ABB RAPID module: 000F2625

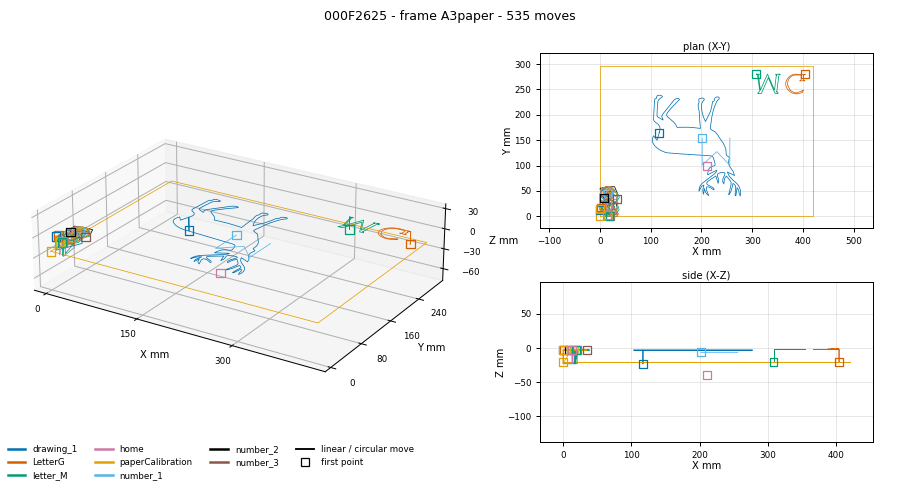
[picture p0: tool path of 000F2625 in frame A3paper, 535 of 535 moves have a stored position in this frame; points joined in program order, loops and branches not executed]
MODULE Module1
	CONST robtarget Target_960:=[[114.097930092,195.477622506,-57.989262096],[0.296983382,-0.000000027,0.000000028,0.954882648],[-1,-1,2,0],[9E+09,9E+09,9E+09,9E+09,9E+09,9E+09]];
	CONST robtarget Target_970:=[[308,280,-20],[1,0,0,0],[0,0,0,0],[9E+09,9E+09,9E+09,9E+09,9E+09,9E+09]];
	CONST robtarget Target_980:=[[308,280,-1],[1,0,0,0],[0,0,0,0],[9E+09,9E+09,9E+09,9E+09,9E+09,9E+09]];
	CONST robtarget Target_990:=[[308,279.6,-1],[1,0,0,0],[0,0,0,0],[9E+09,9E+09,9E+09,9E+09,9E+09,9E+09]];
	CONST robtarget Target_1000:=[[309.6,279.3,-1],[1,0,0,0],[0,0,0,0],[9E+09,9E+09,9E+09,9E+09,9E+09,9E+09]];
	CONST robtarget Target_1010:=[[310.2,278.4,-1],[1,0,0,0],[0,0,0,0],[9E+09,9E+09,9E+09,9E+09,9E+09,9E+09]];
	CONST robtarget Target_1020:=[[314.9,246.9,-1],[1,0,0,0],[0,0,2,0],[9E+09,9E+09,9E+09,9E+09,9E+09,9E+09]];
	CONST robtarget Target_1040:=[[310.75,242.39,-1],[1,0,0,0],[0,0,2,0],[9E+09,9E+09,9E+09,9E+09,9E+09,9E+09]];
	CONST robtarget Target_1050:=[[310.75,241.99,-1],[1,0,0,0],[0,0,0,0],[9E+09,9E+09,9E+09,9E+09,9E+09,9E+09]];
	CONST robtarget Target_1060:=[[317.99,241.99,-1],[1,0,0,0],[0,0,0,0],[9E+09,9E+09,9E+09,9E+09,9E+09,9E+09]];
	CONST robtarget Target_1070:=[[331.45,273.1,-1],[1,0,0,0],[0,0,0,0],[9E+09,9E+09,9E+09,9E+09,9E+09,9E+09]];
	CONST robtarget Target_1080:=[[344.92,241.99,-1],[1,0,0,0],[0,0,0,0],[9E+09,9E+09,9E+09,9E+09,9E+09,9E+09]];
	CONST robtarget Target_1090:=[[351,241.99,-1],[1,0,0,0],[0,0,0,0],[9E+09,9E+09,9E+09,9E+09,9E+09,9E+09]];
	CONST robtarget Target_1100:=[[351,242.39,-1],[1,0,0,0],[0,0,0,0],[9E+09,9E+09,9E+09,9E+09,9E+09,9E+09]];
	CONST robtarget Target_1110:=[[348.2,244.8,-1],[1,0,0,0],[0,0,0,0],[9E+09,9E+09,9E+09,9E+09,9E+09,9E+09]];
	CONST robtarget Target_1120:=[[347.98,246,-1],[1,0,0,0],[0,0,0,0],[9E+09,9E+09,9E+09,9E+09,9E+09,9E+09]];
	CONST robtarget Target_1130:=[[352.51,278,-1],[1,0,0,0],[0,0,0,0],[9E+09,9E+09,9E+09,9E+09,9E+09,9E+09]];
	CONST robtarget Target_1140:=[[353,279,-1],[1,0,0,0],[0,0,0,0],[9E+09,9E+09,9E+09,9E+09,9E+09,9E+09]];
	CONST robtarget Target_1150:=[[354.8,279.7,-1],[1,0,0,0],[0,0,0,0],[9E+09,9E+09,9E+09,9E+09,9E+09,9E+09]];
	CONST robtarget Target_1160:=[[354.8,280,-1],[1,0,0,0],[0,0,0,0],[9E+09,9E+09,9E+09,9E+09,9E+09,9E+09]];
	CONST robtarget Target_1170:=[[346.2,280,-1],[1,0,0,0],[0,0,0,0],[9E+09,9E+09,9E+09,9E+09,9E+09,9E+09]];
	CONST robtarget Target_1180:=[[346.2,279.7,-1],[1,0,0,0],[0,0,0,0],[9E+09,9E+09,9E+09,9E+09,9E+09,9E+09]];
	CONST robtarget Target_1190:=[[347.51,279.3,-1],[1,0,0,0],[0,0,0,0],[9E+09,9E+09,9E+09,9E+09,9E+09,9E+09]];
	CONST robtarget Target_1200:=[[347.96,278,-1],[1,0,0,0],[0,0,0,0],[9E+09,9E+09,9E+09,9E+09,9E+09,9E+09]];
	CONST robtarget Target_1210:=[[343.88,248.52,-1],[1,0,0,0],[0,0,0,0],[9E+09,9E+09,9E+09,9E+09,9E+09,9E+09]];
	CONST robtarget Target_1220:=[[330.1,280,-1],[1,0,0,0],[0,0,0,0],[9E+09,9E+09,9E+09,9E+09,9E+09,9E+09]];
	CONST robtarget Target_1230:=[[329.81,280,-1],[1,0,0,0],[0,0,0,0],[9E+09,9E+09,9E+09,9E+09,9E+09,9E+09]];
	CONST robtarget Target_1240:=[[316.05,248.51,-1],[1,0,0,0],[0,0,0,0],[9E+09,9E+09,9E+09,9E+09,9E+09,9E+09]];
	CONST robtarget Target_1250:=[[312.1,278,-1],[1,0,0,0],[0,0,0,0],[9E+09,9E+09,9E+09,9E+09,9E+09,9E+09]];
	CONST robtarget Target_1260:=[[312.3,279,-1],[1,0,0,0],[0,0,0,0],[9E+09,9E+09,9E+09,9E+09,9E+09,9E+09]];
	CONST robtarget Target_1270:=[[313.8,279.7,-1],[1,0,0,0],[0,0,0,0],[9E+09,9E+09,9E+09,9E+09,9E+09,9E+09]];
	CONST robtarget Target_1280:=[[313.8,280,-1],[1,0,0,0],[0,0,0,0],[9E+09,9E+09,9E+09,9E+09,9E+09,9E+09]];
	CONST robtarget Target_1290:=[[308,280,-1],[1,0,0,0],[0,0,0,0],[9E+09,9E+09,9E+09,9E+09,9E+09,9E+09]];
	CONST robtarget Target_1300:=[[308,280,-20],[1,0,0,0],[0,0,0,0],[9E+09,9E+09,9E+09,9E+09,9E+09,9E+09]];
	CONST robtarget Target_1310:=[[403.47,280,-20],[1,0,0,0],[0,0,0,0],[9E+09,9E+09,9E+09,9E+09,9E+09,9E+09]];
	CONST robtarget Target_1320:=[[403.47,280,-1],[1,0,0,0],[0,0,1,0],[9E+09,9E+09,9E+09,9E+09,9E+09,9E+09]];
	CONST robtarget Target_1330:=[[387,280,-1],[1,0,0,0],[0,0,1,0],[9E+09,9E+09,9E+09,9E+09,9E+09,9E+09]];
	CONST robtarget Target_1340:=[[365.71,260,-1],[1,0,0,0],[0,0,1,0],[9E+09,9E+09,9E+09,9E+09,9E+09,9E+09]];
	CONST robtarget Target_1350:=[[382,241.9,-1],[1,0,0,0],[0,0,1,0],[9E+09,9E+09,9E+09,9E+09,9E+09,9E+09]];
	CONST robtarget Target_1360:=[[387,241.3,-1],[1,0,0,0],[0,0,1,0],[9E+09,9E+09,9E+09,9E+09,9E+09,9E+09]];
	CONST robtarget Target_1370:=[[398.5,244.5,-1],[1,0,0,0],[0,0,1,0],[9E+09,9E+09,9E+09,9E+09,9E+09,9E+09]];
	CONST robtarget Target_1380:=[[400.8,248.26,-1],[1,0,0,0],[0,0,1,0],[9E+09,9E+09,9E+09,9E+09,9E+09,9E+09]];
	CONST robtarget Target_1390:=[[400.4,248.26,-1],[1,0,0,0],[0,0,1,0],[9E+09,9E+09,9E+09,9E+09,9E+09,9E+09]];
	CONST robtarget Target_1400:=[[387,242.79,-1],[1,0,0,0],[0,0,1,0],[9E+09,9E+09,9E+09,9E+09,9E+09,9E+09]];
	CONST robtarget Target_1410:=[[382,244.2,-1],[1,0,0,0],[0,0,1,0],[9E+09,9E+09,9E+09,9E+09,9E+09,9E+09]];
	CONST robtarget Target_1420:=[[370,258,-1],[1,0,0,0],[0,0,1,0],[9E+09,9E+09,9E+09,9E+09,9E+09,9E+09]];
	CONST robtarget Target_1420A:=[[380,272,-1],[1,0,0,0],[0,0,1,0],[9E+09,9E+09,9E+09,9E+09,9E+09,9E+09]];
	CONST robtarget Target_1430:=[[388,278.4,-1],[1,0,0,0],[0,0,1,0],[9E+09,9E+09,9E+09,9E+09,9E+09,9E+09]];
	CONST robtarget Target_1440:=[[392,278.99,-1],[1,0,0,0],[0,0,1,0],[9E+09,9E+09,9E+09,9E+09,9E+09,9E+09]];
	CONST robtarget Target_1450:=[[393,278.75,-1],[1,0,0,0],[0,0,1,0],[9E+09,9E+09,9E+09,9E+09,9E+09,9E+09]];
	CONST robtarget Target_1460:=[[395.8,278,-1],[1,0,0,0],[0,0,1,0],[9E+09,9E+09,9E+09,9E+09,9E+09,9E+09]];
	CONST robtarget Target_1470:=[[396.3,276,-1],[1,0,0,0],[0,0,1,0],[9E+09,9E+09,9E+09,9E+09,9E+09,9E+09]];
	CONST robtarget Target_1480:=[[392.7,278.3,-1],[1,0,0,0],[0,0,1,0],[9E+09,9E+09,9E+09,9E+09,9E+09,9E+09]];
	CONST robtarget Target_1490:=[[395.7,278.2,-1],[1,0,0,0],[0,0,1,0],[9E+09,9E+09,9E+09,9E+09,9E+09,9E+09]];
	CONST robtarget Target_1500:=[[396.3,276,-1],[1,0,0,0],[0,0,1,0],[9E+09,9E+09,9E+09,9E+09,9E+09,9E+09]];
	CONST robtarget Target_1510:=[[396.3,269.1,-1],[1,0,0,0],[0,0,1,0],[9E+09,9E+09,9E+09,9E+09,9E+09,9E+09]];
	CONST robtarget Target_1520:=[[394.9,267.9,-1],[1,0,0,0],[0,0,1,0],[9E+09,9E+09,9E+09,9E+09,9E+09,9E+09]];
	CONST robtarget Target_1530:=[[393.51,267.1,-1],[1,0,0,0],[0,0,1,0],[9E+09,9E+09,9E+09,9E+09,9E+09,9E+09]];
	CONST robtarget Target_1540:=[[393.5,266.8,-1],[1,0,0,0],[0,0,1,0],[9E+09,9E+09,9E+09,9E+09,9E+09,9E+09]];
	CONST robtarget Target_1550:=[[403.5,266.8,-1],[1,0,0,0],[0,0,1,0],[9E+09,9E+09,9E+09,9E+09,9E+09,9E+09]];
	CONST robtarget Target_1560:=[[403.5,267.1,-1],[1,0,0,0],[0,0,1,0],[9E+09,9E+09,9E+09,9E+09,9E+09,9E+09]];
	CONST robtarget Target_1570:=[[401.2,267.9,-1],[1,0,0,0],[0,0,1,0],[9E+09,9E+09,9E+09,9E+09,9E+09,9E+09]];
	CONST robtarget Target_1580:=[[400.8,269.1,-1],[1,0,0,0],[0,0,1,0],[9E+09,9E+09,9E+09,9E+09,9E+09,9E+09]];
	CONST robtarget Target_1590:=[[400.8,276,-1],[1,0,0,0],[0,0,1,0],[9E+09,9E+09,9E+09,9E+09,9E+09,9E+09]];
	CONST robtarget Target_1600:=[[401.2,279,-1],[1,0,0,0],[0,0,1,0],[9E+09,9E+09,9E+09,9E+09,9E+09,9E+09]];
	CONST robtarget Target_1610:=[[403.5,279.7,-1],[1,0,0,0],[0,0,1,0],[9E+09,9E+09,9E+09,9E+09,9E+09,9E+09]];
	CONST robtarget Target_1630:=[[210,100,-40],[1,0,0,0],[0,0,0,0],[9E+09,9E+09,9E+09,9E+09,9E+09,9E+09]];
	CONST robtarget image_startTarget:=[[114.097941212,195.477543406,-3],[0.296983386,0,0,0.954882646],[-1,0,2,0],[9E+09,9E+09,9E+09,9E+09,9E+09,9E+09]];
	CONST robtarget Target_1421:=[[374.2,273.2,-1],[1,0,0,0],[0,0,1,0],[9E+09,9E+09,9E+09,9E+09,9E+09,9E+09]];
	CONST robtarget Target_1411:=[[374.3,249.1,-1],[1,0,0,0],[0,0,1,0],[9E+09,9E+09,9E+09,9E+09,9E+09,9E+09]];
	CONST robtarget Target_1331:=[[370.8,273,-1],[1,0,0,0],[0,0,1,0],[9E+09,9E+09,9E+09,9E+09,9E+09,9E+09]];
	CONST robtarget Target_1341:=[[372.4,247,-1],[1,0,0,0],[0,0,1,0],[9E+09,9E+09,9E+09,9E+09,9E+09,9E+09]];
	CONST robtarget Target_1620:=[[403.5,280,-1],[1,0,0,0],[0,0,1,0],[9E+09,9E+09,9E+09,9E+09,9E+09,9E+09]];
    CONST robtarget Target_2160:=[[193.370337383,219.913130465,-3],[1,0,0,0],[0,0,0,0],[9E+09,9E+09,9E+09,9E+09,9E+09,9E+09]];
    CONST robtarget Target_2190:=[[195.261015335,231.205877786,-3],[1,0,0,0],[0,0,0,0],[9E+09,9E+09,9E+09,9E+09,9E+09,9E+09]];
    CONST robtarget Target_2240:=[[202.476909017,225.935782034,-3],[1,0,0,0],[0,0,0,0],[9E+09,9E+09,9E+09,9E+09,9E+09,9E+09]];
    CONST robtarget Target_2250:=[[200.458270111,222.059210742,-3],[1,0,0,0],[0,0,0,0],[9E+09,9E+09,9E+09,9E+09,9E+09,9E+09]];
    CONST robtarget Target_2260:=[[200.131870923,213.002260799,-3],[1,0,0,0],[0,0,0,0],[9E+09,9E+09,9E+09,9E+09,9E+09,9E+09]];
    CONST robtarget Target_2270:=[[201.352548333,204.144326867,-3],[1,0,0,0],[0,0,0,0],[9E+09,9E+09,9E+09,9E+09,9E+09,9E+09]];
    CONST robtarget Target_2280:=[[203.989899977,195.415486359,-3],[1,0,0,0],[0,0,0,0],[9E+09,9E+09,9E+09,9E+09,9E+09,9E+09]];
    CONST robtarget Target_2310:=[[219.57359463,213.353914551,-3],[1,0,0,0],[0,0,0,0],[9E+09,9E+09,9E+09,9E+09,9E+09,9E+09]];
    CONST robtarget Target_2320:=[[221.72168992,225.083729881,-3],[1,0,0,0],[0,0,0,0],[9E+09,9E+09,9E+09,9E+09,9E+09,9E+09]];
    CONST robtarget Target_2370:=[[226.65209234,233.190693627,-3],[1,0,0,0],[0,0,0,0],[9E+09,9E+09,9E+09,9E+09,9E+09,9E+09]];
    CONST robtarget Target_2440:=[[229.869479521,225.835975339,-3],[1,0,0,0],[0,0,0,0],[9E+09,9E+09,9E+09,9E+09,9E+09,9E+09]];
    CONST robtarget Target_2450:=[[227.167304938,219.606802526,-3],[1,0,0,0],[0,0,0,0],[9E+09,9E+09,9E+09,9E+09,9E+09,9E+09]];
    CONST robtarget Target_2470:=[[220.688053949,197.559828522,-3],[1,0,0,0],[0,0,0,0],[9E+09,9E+09,9E+09,9E+09,9E+09,9E+09]];
    CONST robtarget Target_2490:=[[217.906200407,171.90434605,-3],[1,0,0,0],[0,0,0,0],[9E+09,9E+09,9E+09,9E+09,9E+09,9E+09]];
    CONST robtarget Target_2510:=[[227.578391856,165.853990796,-3],[1,0,0,0],[0,0,0,0],[9E+09,9E+09,9E+09,9E+09,9E+09,9E+09]];
    CONST robtarget Target_2520:=[[232.79626775,159.200927161,-3],[1,0,0,0],[0,0,0,0],[9E+09,9E+09,9E+09,9E+09,9E+09,9E+09]];
    CONST robtarget Target_2530:=[[235.197557217,154.8951234,-3],[1,0,0,0],[0,0,0,0],[9E+09,9E+09,9E+09,9E+09,9E+09,9E+09]];
    CONST robtarget Target_2560:=[[248.128216692,130.946667408,-3],[1,0,0,0],[0,0,0,0],[9E+09,9E+09,9E+09,9E+09,9E+09,9E+09]];
    CONST robtarget Target_2580:=[[249.072498858,120.410096923,-3],[1,0,0,0],[0,0,0,0],[9E+09,9E+09,9E+09,9E+09,9E+09,9E+09]];
    CONST robtarget Target_2590:=[[251.497695182,118.536506038,-3],[1,0,0,0],[0,0,0,0],[9E+09,9E+09,9E+09,9E+09,9E+09,9E+09]];
    CONST robtarget Target_2610:=[[254.693387483,115.452076001,-3],[1,0,0,0],[0,0,0,0],[9E+09,9E+09,9E+09,9E+09,9E+09,9E+09]];
    CONST robtarget Target_2660:=[[265.141029781,80.351141961,-3],[1,0,0,0],[0,0,0,0],[9E+09,9E+09,9E+09,9E+09,9E+09,9E+09]];
    CONST robtarget Target_2680:=[[253.43619882,81.678122788,-3],[1,0,0,0],[0,0,0,0],[9E+09,9E+09,9E+09,9E+09,9E+09,9E+09]];
    CONST robtarget Target_2690:=[[256.347942609,77.175605659,-3],[1,0,0,0],[0,0,0,0],[9E+09,9E+09,9E+09,9E+09,9E+09,9E+09]];
    CONST robtarget Target_2710:=[[267.614835775,66.494604603,-3],[1,0,0,0],[0,0,0,0],[9E+09,9E+09,9E+09,9E+09,9E+09,9E+09]];
    CONST robtarget Target_2720:=[[271.684226977,62.292746796,-3],[1,0,0,0],[0,0,0,0],[9E+09,9E+09,9E+09,9E+09,9E+09,9E+09]];
    CONST robtarget Target_2730:=[[274.598698271,57.568830631,-3],[1,0,0,0],[0,0,0,0],[9E+09,9E+09,9E+09,9E+09,9E+09,9E+09]];
    CONST robtarget Target_2740:=[[276.417527718,52.342499268,-3],[1,0,0,0],[0,0,0,0],[9E+09,9E+09,9E+09,9E+09,9E+09,9E+09]];
    CONST robtarget Target_2750:=[[277.199993374,46.633395866,-3],[1,0,0,0],[0,0,0,0],[9E+09,9E+09,9E+09,9E+09,9E+09,9E+09]];
    CONST robtarget Target_2760:=[[276.903780142,43.337729466,-3],[1,0,0,0],[0,0,0,0],[9E+09,9E+09,9E+09,9E+09,9E+09,9E+09]];
    CONST robtarget Target_2770:=[[276.283936631,40.026597635,-3],[1,0,0,0],[0,0,0,0],[9E+09,9E+09,9E+09,9E+09,9E+09,9E+09]];
    CONST robtarget Target_2780:=[[274.453452076,43.865061405,-3],[1,0,0,0],[0,0,0,0],[9E+09,9E+09,9E+09,9E+09,9E+09,9E+09]];
    CONST robtarget Target_2790:=[[273.824145046,48.089825742,-3],[1,0,0,0],[0,0,0,0],[9E+09,9E+09,9E+09,9E+09,9E+09,9E+09]];
    CONST robtarget Target_2810:=[[270.016935967,56.440062852,-3],[1,0,0,0],[0,0,0,0],[9E+09,9E+09,9E+09,9E+09,9E+09,9E+09]];
    CONST robtarget Target_2820:=[[267.749530853,40.667201266,-3],[1,0,0,0],[0,0,0,0],[9E+09,9E+09,9E+09,9E+09,9E+09,9E+09]];
    CONST robtarget Target_2830:=[[266.302922269,40.756977809,-3],[1,0,0,0],[0,0,0,0],[9E+09,9E+09,9E+09,9E+09,9E+09,9E+09]];
    CONST robtarget Target_2840:=[[266.441249646,47.650430951,-3],[1,0,0,0],[0,0,0,0],[9E+09,9E+09,9E+09,9E+09,9E+09,9E+09]];
    CONST robtarget Target_2850:=[[267.430396017,57.809270006,-3],[1,0,0,0],[0,0,0,0],[9E+09,9E+09,9E+09,9E+09,9E+09,9E+09]];
    CONST robtarget Target_2860:=[[266.669716785,60.560651269,-3],[1,0,0,0],[0,0,0,0],[9E+09,9E+09,9E+09,9E+09,9E+09,9E+09]];
    CONST robtarget Target_2870:=[[264.903208645,62.848641641,-3],[1,0,0,0],[0,0,0,0],[9E+09,9E+09,9E+09,9E+09,9E+09,9E+09]];
    CONST robtarget Target_2880:=[[262.176964385,64.847561878,-3],[1,0,0,0],[0,0,0,0],[9E+09,9E+09,9E+09,9E+09,9E+09,9E+09]];
    CONST robtarget Target_2890:=[[259.299549793,53.075582965,-3],[1,0,0,0],[0,0,0,0],[9E+09,9E+09,9E+09,9E+09,9E+09,9E+09]];
    CONST robtarget Target_2910:=[[253.896826863,42.44360071,-3],[1,0,0,0],[0,0,0,0],[9E+09,9E+09,9E+09,9E+09,9E+09,9E+09]];
    CONST robtarget Target_2920:=[[253.921604349,44.335351342,-3],[1,0,0,0],[0,0,0,0],[9E+09,9E+09,9E+09,9E+09,9E+09,9E+09]];
    CONST robtarget Target_2930:=[[258.274708163,62.583521728,-3],[1,0,0,0],[0,0,0,0],[9E+09,9E+09,9E+09,9E+09,9E+09,9E+09]];
    CONST robtarget Target_2940:=[[258.451861421,65.72308068,-3],[1,0,0,0],[0,0,0,0],[9E+09,9E+09,9E+09,9E+09,9E+09,9E+09]];
    CONST robtarget Target_2950:=[[257.604969868,68.580619068,-3],[1,0,0,0],[0,0,0,0],[9E+09,9E+09,9E+09,9E+09,9E+09,9E+09]];
    CONST robtarget Target_2960:=[[253.567432927,74.071600383,-3],[1,0,0,0],[0,0,0,0],[9E+09,9E+09,9E+09,9E+09,9E+09,9E+09]];
    CONST robtarget Target_2970:=[[249.243881242,79.371580046,-3],[1,0,0,0],[0,0,0,0],[9E+09,9E+09,9E+09,9E+09,9E+09,9E+09]];
    CONST robtarget Target_2980:=[[246.352038922,75.978183413,-3],[1,0,0,0],[0,0,0,0],[9E+09,9E+09,9E+09,9E+09,9E+09,9E+09]];
    CONST robtarget Target_2990:=[[244.977183436,72.142467996,-3],[1,0,0,0],[0,0,0,0],[9E+09,9E+09,9E+09,9E+09,9E+09,9E+09]];
    CONST robtarget Target_3010:=[[242.513799023,66.424388789,-3],[1,0,0,0],[0,0,0,0],[9E+09,9E+09,9E+09,9E+09,9E+09,9E+09]];
    CONST robtarget Target_3030:=[[242.453890553,75.021110222,-3],[1,0,0,0],[0,0,0,0],[9E+09,9E+09,9E+09,9E+09,9E+09,9E+09]];
    CONST robtarget Target_3040:=[[245.184309174,80.346921596,-3],[1,0,0,0],[0,0,0,0],[9E+09,9E+09,9E+09,9E+09,9E+09,9E+09]];
    CONST robtarget Target_3050:=[[246.355111707,84.063986783,-3],[1,0,0,0],[0,0,0,0],[9E+09,9E+09,9E+09,9E+09,9E+09,9E+09]];
    CONST robtarget Target_3060:=[[245.799291444,85.605935054,-3],[1,0,0,0],[0,0,0,0],[9E+09,9E+09,9E+09,9E+09,9E+09,9E+09]];
    CONST robtarget Target_3070:=[[243.989820642,86.456427668,-3],[1,0,0,0],[0,0,0,0],[9E+09,9E+09,9E+09,9E+09,9E+09,9E+09]];
    CONST robtarget Target_3080:=[[238.686656522,86.356933008,-3],[1,0,0,0],[0,0,0,0],[9E+09,9E+09,9E+09,9E+09,9E+09,9E+09]];
    CONST robtarget Target_3090:=[[233.626373536,84.723508323,-3],[1,0,0,0],[0,0,0,0],[9E+09,9E+09,9E+09,9E+09,9E+09,9E+09]];
    CONST robtarget Target_3110:=[[231.229705834,80.92138457,-3],[1,0,0,0],[0,0,0,0],[9E+09,9E+09,9E+09,9E+09,9E+09,9E+09]];
    CONST robtarget Target_3120:=[[232.687410286,76.08625905,-3],[1,0,0,0],[0,0,0,0],[9E+09,9E+09,9E+09,9E+09,9E+09,9E+09]];
    CONST robtarget Target_3130:=[[233.844814545,70.463867465,-3],[1,0,0,0],[0,0,0,0],[9E+09,9E+09,9E+09,9E+09,9E+09,9E+09]];
    CONST robtarget Target_3140:=[[232.683868526,64.986793847,-3],[1,0,0,0],[0,0,0,0],[9E+09,9E+09,9E+09,9E+09,9E+09,9E+09]];
    CONST robtarget Target_3150:=[[228.374978172,79.484110725,-3],[1,0,0,0],[0,0,0,0],[9E+09,9E+09,9E+09,9E+09,9E+09,9E+09]];
    CONST robtarget Target_3160:=[[219.965736687,74.015207284,-3],[1,0,0,0],[0,0,0,0],[9E+09,9E+09,9E+09,9E+09,9E+09,9E+09]];
    CONST robtarget Target_3170:=[[212.554359432,68.787624505,-3],[1,0,0,0],[0,0,0,0],[9E+09,9E+09,9E+09,9E+09,9E+09,9E+09]];
    CONST robtarget Target_3180:=[[210.677030599,66.626673914,-3],[1,0,0,0],[0,0,0,0],[9E+09,9E+09,9E+09,9E+09,9E+09,9E+09]];
    CONST robtarget Target_3190:=[[210.38708356,64.517394422,-3],[1,0,0,0],[0,0,0,0],[9E+09,9E+09,9E+09,9E+09,9E+09,9E+09]];
    CONST robtarget Target_3210:=[[214.11130813,61.047061647,-3],[1,0,0,0],[0,0,0,0],[9E+09,9E+09,9E+09,9E+09,9E+09,9E+09]];
    CONST robtarget Target_3220:=[[222.416533213,56.844968834,-3],[1,0,0,0],[0,0,0,0],[9E+09,9E+09,9E+09,9E+09,9E+09,9E+09]];
    CONST robtarget Target_3230:=[[223.832262364,55.151481233,-3],[1,0,0,0],[0,0,0,0],[9E+09,9E+09,9E+09,9E+09,9E+09,9E+09]];
    CONST robtarget Target_3240:=[[224.991497966,53.059964778,-3],[1,0,0,0],[0,0,0,0],[9E+09,9E+09,9E+09,9E+09,9E+09,9E+09]];
    CONST robtarget Target_3260:=[[217.660699108,56.478310873,-3],[1,0,0,0],[0,0,0,0],[9E+09,9E+09,9E+09,9E+09,9E+09,9E+09]];
    CONST robtarget Target_3270:=[[214.198336017,57.976316513,-3],[1,0,0,0],[0,0,0,0],[9E+09,9E+09,9E+09,9E+09,9E+09,9E+09]];
    CONST robtarget Target_3280:=[[210.117558581,57.951519862,-3],[1,0,0,0],[0,0,0,0],[9E+09,9E+09,9E+09,9E+09,9E+09,9E+09]];
    CONST robtarget Target_3290:=[[209.641800543,53.313049599,-3],[1,0,0,0],[0,0,0,0],[9E+09,9E+09,9E+09,9E+09,9E+09,9E+09]];
    CONST robtarget Target_3310:=[[214.391838304,40.955022791,-3],[1,0,0,0],[0,0,0,0],[9E+09,9E+09,9E+09,9E+09,9E+09,9E+09]];
    CONST robtarget Target_3320:=[[210.799968866,43.482482486,-3],[1,0,0,0],[0,0,0,0],[9E+09,9E+09,9E+09,9E+09,9E+09,9E+09]];
    CONST robtarget Target_3330:=[[208.378326367,46.710824702,-3],[1,0,0,0],[0,0,0,0],[9E+09,9E+09,9E+09,9E+09,9E+09,9E+09]];
    CONST robtarget Target_3340:=[[205.519567882,54.640553293,-3],[1,0,0,0],[0,0,0,0],[9E+09,9E+09,9E+09,9E+09,9E+09,9E+09]];
    CONST robtarget Target_3350:=[[204.274957824,43.449915608,-3],[1,0,0,0],[0,0,0,0],[9E+09,9E+09,9E+09,9E+09,9E+09,9E+09]];
    CONST robtarget Target_3360:=[[202.779864784,47.961332689,-3],[1,0,0,0],[0,0,0,0],[9E+09,9E+09,9E+09,9E+09,9E+09,9E+09]];
    CONST robtarget Target_3370:=[[202.686470534,52.473353811,-3],[1,0,0,0],[0,0,0,0],[9E+09,9E+09,9E+09,9E+09,9E+09,9E+09]];
    CONST robtarget Target_3380:=[[204.779738543,61.691960466,-3],[1,0,0,0],[0,0,0,0],[9E+09,9E+09,9E+09,9E+09,9E+09,9E+09]];
    CONST robtarget Target_3390:=[[200.828885863,59.46054831,-3],[1,0,0,0],[0,0,0,0],[9E+09,9E+09,9E+09,9E+09,9E+09,9E+09]];
    CONST robtarget Target_3410:=[[195.145559108,49.337942562,-3],[1,0,0,0],[0,0,0,0],[9E+09,9E+09,9E+09,9E+09,9E+09,9E+09]];
    CONST robtarget Target_3420:=[[195.353663461,54.280625926,-3],[1,0,0,0],[0,0,0,0],[9E+09,9E+09,9E+09,9E+09,9E+09,9E+09]];
    CONST robtarget Target_3430:=[[196.676958422,58.695618887,-3],[1,0,0,0],[0,0,0,0],[9E+09,9E+09,9E+09,9E+09,9E+09,9E+09]];
    CONST robtarget Target_3440:=[[199.103095305,62.59104984,-3],[1,0,0,0],[0,0,0,0],[9E+09,9E+09,9E+09,9E+09,9E+09,9E+09]];
    CONST robtarget Target_3450:=[[202.619725421,65.975047185,-3],[1,0,0,0],[0,0,0,0],[9E+09,9E+09,9E+09,9E+09,9E+09,9E+09]];
    CONST robtarget Target_3470:=[[228.146134612,86.522665975,-3],[1,0,0,0],[0,0,0,0],[9E+09,9E+09,9E+09,9E+09,9E+09,9E+09]];
    CONST robtarget Target_3480:=[[230.400867961,89.633137216,-3],[1,0,0,0],[0,0,0,0],[9E+09,9E+09,9E+09,9E+09,9E+09,9E+09]];
    CONST robtarget Target_3490:=[[229.502924222,90.649093077,-3],[1,0,0,0],[0,0,0,0],[9E+09,9E+09,9E+09,9E+09,9E+09,9E+09]];
    CONST robtarget Target_3510:=[[213.02947803,88.518895223,-3],[1,0,0,0],[0,0,0,0],[9E+09,9E+09,9E+09,9E+09,9E+09,9E+09]];
    CONST robtarget Target_3520:=[[214.278806706,92.822596592,-3],[1,0,0,0],[0,0,0,0],[9E+09,9E+09,9E+09,9E+09,9E+09,9E+09]];
    CONST robtarget Target_3530:=[[216.417539352,95.955068284,-3],[1,0,0,0],[0,0,0,0],[9E+09,9E+09,9E+09,9E+09,9E+09,9E+09]];
    CONST robtarget Target_3540:=[[219.585437503,98.050973568,-3],[1,0,0,0],[0,0,0,0],[9E+09,9E+09,9E+09,9E+09,9E+09,9E+09]];
    CONST robtarget Target_3550:=[[223.922262697,99.244975714,-3],[1,0,0,0],[0,0,0,0],[9E+09,9E+09,9E+09,9E+09,9E+09,9E+09]];
    CONST robtarget Target_3560:=[[226.759287881,100.694337329,-3],[1,0,0,0],[0,0,0,0],[9E+09,9E+09,9E+09,9E+09,9E+09,9E+09]];
    CONST robtarget Target_3570:=[[226.681756776,103.944262165,-3],[1,0,0,0],[0,0,0,0],[9E+09,9E+09,9E+09,9E+09,9E+09,9E+09]];
    CONST robtarget Target_3580:=[[224.505103701,112.138872075,-3],[1,0,0,0],[0,0,0,0],[9E+09,9E+09,9E+09,9E+09,9E+09,9E+09]];
    CONST robtarget Target_3590:=[[223.414408001,115.469817817,-3],[1,0,0,0],[0,0,0,0],[9E+09,9E+09,9E+09,9E+09,9E+09,9E+09]];
    CONST robtarget Target_3610:=[[219.460026303,118.825512034,-3],[1,0,0,0],[0,0,0,0],[9E+09,9E+09,9E+09,9E+09,9E+09,9E+09]];
    CONST robtarget Target_3620:=[[215.936165455,119.356824487,-3],[1,0,0,0],[0,0,0,0],[9E+09,9E+09,9E+09,9E+09,9E+09,9E+09]];
    CONST robtarget Target_3630:=[[155.66830507,123.260946897,-3],[1,0,0,0],[0,0,0,0],[9E+09,9E+09,9E+09,9E+09,9E+09,9E+09]];
    CONST robtarget Target_3640:=[[133.585682803,125.008606143,-3],[1,0,0,0],[0,0,0,0],[9E+09,9E+09,9E+09,9E+09,9E+09,9E+09]];
    CONST robtarget Target_3650:=[[128.099986881,126.297578543,-3],[1,0,0,0],[0,0,0,0],[9E+09,9E+09,9E+09,9E+09,9E+09,9E+09]];
    CONST robtarget Target_3660:=[[122.770725675,128.44117716,-3],[1,0,0,0],[0,0,0,0],[9E+09,9E+09,9E+09,9E+09,9E+09,9E+09]];
    CONST robtarget Target_3670:=[[118.375825136,130.605132148,-3],[1,0,0,0],[0,0,0,0],[9E+09,9E+09,9E+09,9E+09,9E+09,9E+09]];
    CONST robtarget Target_3680:=[[114.276287738,133.278163879,-3],[1,0,0,0],[0,0,0,0],[9E+09,9E+09,9E+09,9E+09,9E+09,9E+09]];
    CONST robtarget Target_3690:=[[108.31401898,138.447566871,-3],[1,0,0,0],[0,0,0,0],[9E+09,9E+09,9E+09,9E+09,9E+09,9E+09]];
    CONST robtarget Target_3710:=[[103.212048819,150.747792156,-3],[1,0,0,0],[0,0,0,0],[9E+09,9E+09,9E+09,9E+09,9E+09,9E+09]];
    CONST robtarget Target_3720:=[[103.919723158,154.520288699,-3],[1,0,0,0],[0,0,0,0],[9E+09,9E+09,9E+09,9E+09,9E+09,9E+09]];
    CONST robtarget Target_3730:=[[105.613280939,158.670782312,-3],[1,0,0,0],[0,0,0,0],[9E+09,9E+09,9E+09,9E+09,9E+09,9E+09]];
    CONST robtarget Target_3740:=[[112.529465698,149.875319719,-3],[1,0,0,0],[0,0,0,0],[9E+09,9E+09,9E+09,9E+09,9E+09,9E+09]];
    CONST robtarget Target_3750:=[[116.864395565,164.59256718,-3],[1,0,0,0],[0,0,0,0],[9E+09,9E+09,9E+09,9E+09,9E+09,9E+09]];
    CONST robtarget Target_1860:=[[112.780653432,197.331638937,-3],[1,0,0,0],[0,0,0,0],[9E+09,9E+09,9E+09,9E+09,9E+09,9E+09]];
    CONST robtarget Target_2080:=[[152.038829652,175.1593366,-3],[1,0,0,0],[0,0,0,0],[9E+09,9E+09,9E+09,9E+09,9E+09,9E+09]];
    CONST robtarget Target_3020:=[[241.726872614,69.136971847,-3],[1,0,0,0],[0,0,0,0],[9E+09,9E+09,9E+09,9E+09,9E+09,9E+09]];
    CONST robtarget Target_2640:=[[255.55352801,98.15492303,-3],[1,0,0,0],[0,0,0,0],[9E+09,9E+09,9E+09,9E+09,9E+09,9E+09]];
    CONST robtarget Target_2120:=[[197.917101799,173.183120269,-3],[1,0,0,0],[0,0,0,0],[9E+09,9E+09,9E+09,9E+09,9E+09,9E+09]];
    CONST robtarget Target_1850:=[[112.322584565,199.686358994,-3],[1,0,0,0],[0,0,0,0],[9E+09,9E+09,9E+09,9E+09,9E+09,9E+09]];
    CONST robtarget Target_1930:=[[124.987181965,202.815326796,-3],[1,0,0,0],[0,0,0,0],[9E+09,9E+09,9E+09,9E+09,9E+09,9E+09]];
    CONST robtarget Target_1760:=[[113.175108389,237.881718509,-3],[1,0,0,0],[0,0,0,0],[9E+09,9E+09,9E+09,9E+09,9E+09,9E+09]];
    CONST robtarget Target_2570:=[[248.603313012,123.194262198,-3],[1,0,0,0],[0,0,0,0],[9E+09,9E+09,9E+09,9E+09,9E+09,9E+09]];
    CONST robtarget Target_1940:=[[146.479851245,229.690888833,-3],[1,0,0,0],[0,0,0,0],[9E+09,9E+09,9E+09,9E+09,9E+09,9E+09]];
    CONST robtarget Target_1890:=[[124.588660422,189.645922432,-3],[1,0,0,0],[0,0,0,0],[9E+09,9E+09,9E+09,9E+09,9E+09,9E+09]];
    CONST robtarget Target_1990:=[[143.386028726,216.472160161,-3],[1,0,0,0],[0,0,0,0],[9E+09,9E+09,9E+09,9E+09,9E+09,9E+09]];
    CONST robtarget Target_1960:=[[153.996438131,232.359045465,-3],[1,0,0,0],[0,0,0,0],[9E+09,9E+09,9E+09,9E+09,9E+09,9E+09]];
    CONST robtarget Target_1920:=[[122.033123429,198.293656571,-3],[1,0,0,0],[0,0,0,0],[9E+09,9E+09,9E+09,9E+09,9E+09,9E+09]];
    CONST robtarget Target_1970:=[[155.686057122,231.358602968,-3],[1,0,0,0],[0,0,0,0],[9E+09,9E+09,9E+09,9E+09,9E+09,9E+09]];
    CONST robtarget Target_1640:=[[116.864395565,164.59256718,-3],[1,0,0,0],[0,0,0,0],[9E+09,9E+09,9E+09,9E+09,9E+09,9E+09]];
    CONST robtarget Target_1700:=[[105.460399665,190.998170229,-3],[1,0,0,0],[0,0,0,0],[9E+09,9E+09,9E+09,9E+09,9E+09,9E+09]];
    CONST robtarget Target_1800:=[[122.788239246,235.080918952,-3],[1,0,0,0],[0,0,0,0],[9E+09,9E+09,9E+09,9E+09,9E+09,9E+09]];
    CONST robtarget Target_1900:=[[123.322560124,193.264620662,-3],[1,0,0,0],[0,0,0,0],[9E+09,9E+09,9E+09,9E+09,9E+09,9E+09]];
    CONST robtarget Target_2000:=[[138.216503942,210.589237829,-3],[1,0,0,0],[0,0,0,0],[9E+09,9E+09,9E+09,9E+09,9E+09,9E+09]];
    CONST robtarget Target_2100:=[[175.283029198,175.465591704,-3],[1,0,0,0],[0,0,0,0],[9E+09,9E+09,9E+09,9E+09,9E+09,9E+09]];
    CONST robtarget Target_2200:=[[197.204607445,232.112473887,-3],[1,0,0,0],[0,0,0,0],[9E+09,9E+09,9E+09,9E+09,9E+09,9E+09]];
    CONST robtarget Target_2300:=[[216.653373158,204.262410012,-3],[1,0,0,0],[0,0,0,0],[9E+09,9E+09,9E+09,9E+09,9E+09,9E+09]];
    CONST robtarget Target_2400:=[[234.529319608,234.44032996,-3],[1,0,0,0],[0,0,0,0],[9E+09,9E+09,9E+09,9E+09,9E+09,9E+09]];
    CONST robtarget Target_2500:=[[220.374264807,170.158152985,-3],[1,0,0,0],[0,0,0,0],[9E+09,9E+09,9E+09,9E+09,9E+09,9E+09]];
    CONST robtarget Target_2600:=[[253.646962041,117.233560169,-3],[1,0,0,0],[0,0,0,0],[9E+09,9E+09,9E+09,9E+09,9E+09,9E+09]];
    CONST robtarget Target_2700:=[[260.733890497,72.527955155,-3],[1,0,0,0],[0,0,0,0],[9E+09,9E+09,9E+09,9E+09,9E+09,9E+09]];
    CONST robtarget Target_2800:=[[272.857983642,52.38634233,-3],[1,0,0,0],[0,0,0,0],[9E+09,9E+09,9E+09,9E+09,9E+09,9E+09]];
    CONST robtarget Target_2900:=[[257.242449633,47.510621314,-3],[1,0,0,0],[0,0,0,0],[9E+09,9E+09,9E+09,9E+09,9E+09,9E+09]];
    CONST robtarget Target_3000:=[[244.096850582,63.785944421,-3],[1,0,0,0],[0,0,0,0],[9E+09,9E+09,9E+09,9E+09,9E+09,9E+09]];
    CONST robtarget Target_3100:=[[231.743913616,83.0482726,-3],[1,0,0,0],[0,0,0,0],[9E+09,9E+09,9E+09,9E+09,9E+09,9E+09]];
    CONST robtarget Target_3200:=[[211.570011631,62.608089257,-3],[1,0,0,0],[0,0,0,0],[9E+09,9E+09,9E+09,9E+09,9E+09,9E+09]];
    CONST robtarget Target_3300:=[[210.858980805,49.109132371,-3],[1,0,0,0],[0,0,0,0],[9E+09,9E+09,9E+09,9E+09,9E+09,9E+09]];
    CONST robtarget Target_3400:=[[198.474872074,56.293554813,-3],[1,0,0,0],[0,0,0,0],[9E+09,9E+09,9E+09,9E+09,9E+09,9E+09]];
    CONST robtarget Target_3500:=[[212.02612724,81.765033631,-3],[1,0,0,0],[0,0,0,0],[9E+09,9E+09,9E+09,9E+09,9E+09,9E+09]];
    CONST robtarget Target_3600:=[[221.842744676,117.614270474,-3],[1,0,0,0],[0,0,0,0],[9E+09,9E+09,9E+09,9E+09,9E+09,9E+09]];
    CONST robtarget Target_3700:=[[104.369117087,144.13874832,-3],[1,0,0,0],[0,0,0,0],[9E+09,9E+09,9E+09,9E+09,9E+09,9E+09]];
    CONST robtarget Target_3250:=[[224.035720598,52.221180493,-3],[1,0,0,0],[0,0,0,0],[9E+09,9E+09,9E+09,9E+09,9E+09,9E+09]];
    CONST robtarget Target_3460:=[[225.626513676,83.742579114,-3],[1,0,0,0],[0,0,0,0],[9E+09,9E+09,9E+09,9E+09,9E+09,9E+09]];
    CONST robtarget Target_1830:=[[114.238061027,226.869080325,-3],[1,0,0,0],[0,0,0,0],[9E+09,9E+09,9E+09,9E+09,9E+09,9E+09]];
    CONST robtarget Target_2210:=[[202.154560124,233.036660078,-3],[1,0,0,0],[0,0,0,0],[9E+09,9E+09,9E+09,9E+09,9E+09,9E+09]];
    CONST robtarget Target_2050:=[[134.760341735,194.66375866,-3],[1,0,0,0],[0,0,0,0],[9E+09,9E+09,9E+09,9E+09,9E+09,9E+09]];
    CONST robtarget Target_2410:=[[234.96018158,232.530608383,-3],[1,0,0,0],[0,0,0,0],[9E+09,9E+09,9E+09,9E+09,9E+09,9E+09]];
    CONST robtarget Target_1770:=[[116.657845409,238.688158697,-3],[1,0,0,0],[0,0,0,0],[9E+09,9E+09,9E+09,9E+09,9E+09,9E+09]];
    CONST robtarget Target_1780:=[[119.796419517,237.931449366,-3],[1,0,0,0],[0,0,0,0],[9E+09,9E+09,9E+09,9E+09,9E+09,9E+09]];
    CONST robtarget Target_2110:=[[186.710846358,174.487070224,-3],[1,0,0,0],[0,0,0,0],[9E+09,9E+09,9E+09,9E+09,9E+09,9E+09]];
    CONST robtarget Target_2670:=[[250.977865837,87.276073215,-3],[1,0,0,0],[0,0,0,0],[9E+09,9E+09,9E+09,9E+09,9E+09,9E+09]];
    CONST robtarget Target_1710:=[[107.647683143,228.882143819,-3],[1,0,0,0],[0,0,0,0],[9E+09,9E+09,9E+09,9E+09,9E+09,9E+09]];
    CONST robtarget Target_1980:=[[156.805532081,230.035294909,-3],[1,0,0,0],[0,0,0,0],[9E+09,9E+09,9E+09,9E+09,9E+09,9E+09]];
    CONST robtarget Target_2460:=[[223.235919709,208.723836407,-3],[1,0,0,0],[0,0,0,0],[9E+09,9E+09,9E+09,9E+09,9E+09,9E+09]];
    CONST robtarget Target_2290:=[[207.913523491,186.74581669,-3],[1,0,0,0],[0,0,0,0],[9E+09,9E+09,9E+09,9E+09,9E+09,9E+09]];
    CONST robtarget Target_2040:=[[132.427776836,196.983355,-3],[1,0,0,0],[0,0,0,0],[9E+09,9E+09,9E+09,9E+09,9E+09,9E+09]];
    CONST robtarget Target_2230:=[[205.725967473,229.920852791,-3],[1,0,0,0],[0,0,0,0],[9E+09,9E+09,9E+09,9E+09,9E+09,9E+09]];
    CONST robtarget Target_2010:=[[133.33629989,204.46386732,-3],[1,0,0,0],[0,0,0,0],[9E+09,9E+09,9E+09,9E+09,9E+09,9E+09]];
    CONST robtarget Target_2170:=[[195.312357648,224.265300055,-3],[1,0,0,0],[0,0,0,0],[9E+09,9E+09,9E+09,9E+09,9E+09,9E+09]];
    CONST robtarget Target_1950:=[[149.825529864,231.592090096,-3],[1,0,0,0],[0,0,0,0],[9E+09,9E+09,9E+09,9E+09,9E+09,9E+09]];
    CONST robtarget Target_2030:=[[131.39673452,199.241626041,-3],[1,0,0,0],[0,0,0,0],[9E+09,9E+09,9E+09,9E+09,9E+09,9E+09]];
    CONST robtarget Target_2650:=[[262.260780735,88.499919006,-3],[1,0,0,0],[0,0,0,0],[9E+09,9E+09,9E+09,9E+09,9E+09,9E+09]];
    CONST robtarget Target_1650:=[[118.45535758,171.519585957,-3],[1,0,0,0],[0,0,0,0],[9E+09,9E+09,9E+09,9E+09,9E+09,9E+09]];
    CONST robtarget Target_1730:=[[110.146848112,231.469472758,-3],[1,0,0,0],[0,0,0,0],[9E+09,9E+09,9E+09,9E+09,9E+09,9E+09]];
    CONST robtarget Target_1660:=[[117.790934909,176.903449933,-3],[1,0,0,0],[0,0,0,0],[9E+09,9E+09,9E+09,9E+09,9E+09,9E+09]];
    CONST robtarget Target_1750:=[[111.2939973,234.524441753,-3],[1,0,0,0],[0,0,0,0],[9E+09,9E+09,9E+09,9E+09,9E+09,9E+09]];
    CONST robtarget Target_1820:=[[115.692304632,229.503383528,-3],[1,0,0,0],[0,0,0,0],[9E+09,9E+09,9E+09,9E+09,9E+09,9E+09]];
    CONST robtarget Target_2350:=[[225.115772308,227.80250181,-3],[1,0,0,0],[0,0,0,0],[9E+09,9E+09,9E+09,9E+09,9E+09,9E+09]];
    CONST robtarget Target_1790:=[[122.9153456,236.720407396,-3],[1,0,0,0],[0,0,0,0],[9E+09,9E+09,9E+09,9E+09,9E+09,9E+09]];
    CONST robtarget Target_2620:=[[253.348083173,107.107874674,-3],[1,0,0,0],[0,0,0,0],[9E+09,9E+09,9E+09,9E+09,9E+09,9E+09]];
    CONST robtarget Target_2130:=[[196.442051112,190.161844469,-3],[1,0,0,0],[0,0,0,0],[9E+09,9E+09,9E+09,9E+09,9E+09,9E+09]];
    CONST robtarget Target_2360:=[[225.378464694,230.938198082,-3],[1,0,0,0],[0,0,0,0],[9E+09,9E+09,9E+09,9E+09,9E+09,9E+09]];
    CONST robtarget Target_2540:=[[242.460261055,144.622396077,-3],[1,0,0,0],[0,0,0,0],[9E+09,9E+09,9E+09,9E+09,9E+09,9E+09]];
    CONST robtarget Target_2480:=[[217.424368094,174.847257691,-3],[1,0,0,0],[0,0,0,0],[9E+09,9E+09,9E+09,9E+09,9E+09,9E+09]];
    CONST robtarget Target_2180:=[[194.650640534,229.679693651,-3],[1,0,0,0],[0,0,0,0],[9E+09,9E+09,9E+09,9E+09,9E+09,9E+09]];
    CONST robtarget Target_2020:=[[131.69148535,201.660990557,-3],[1,0,0,0],[0,0,0,0],[9E+09,9E+09,9E+09,9E+09,9E+09,9E+09]];
    CONST robtarget Target_2630:=[[253.961161866,102.533093992,-3],[1,0,0,0],[0,0,0,0],[9E+09,9E+09,9E+09,9E+09,9E+09,9E+09]];
    CONST robtarget Target_2220:=[[204.28233594,232.378888522,-3],[1,0,0,0],[0,0,0,0],[9E+09,9E+09,9E+09,9E+09,9E+09,9E+09]];
    CONST robtarget Target_1880:=[[118.928304574,192.620188811,-3],[1,0,0,0],[0,0,0,0],[9E+09,9E+09,9E+09,9E+09,9E+09,9E+09]];
    CONST robtarget Target_2330:=[[222.213480929,226.375232188,-3],[1,0,0,0],[0,0,0,0],[9E+09,9E+09,9E+09,9E+09,9E+09,9E+09]];
    CONST robtarget Target_1690:=[[106.492973467,187.973742876,-3],[1,0,0,0],[0,0,0,0],[9E+09,9E+09,9E+09,9E+09,9E+09,9E+09]];
    CONST robtarget Target_1840:=[[113.075917318,213.295728508,-3],[1,0,0,0],[0,0,0,0],[9E+09,9E+09,9E+09,9E+09,9E+09,9E+09]];
    CONST robtarget Target_2140:=[[195.443614009,206.901455071,-3],[1,0,0,0],[0,0,0,0],[9E+09,9E+09,9E+09,9E+09,9E+09,9E+09]];
    CONST robtarget Target_2390:=[[232.123329048,235.32552252,-3],[1,0,0,0],[0,0,0,0],[9E+09,9E+09,9E+09,9E+09,9E+09,9E+09]];
    CONST robtarget Target_2060:=[[144.978412323,185.8937717,-3],[1,0,0,0],[0,0,0,0],[9E+09,9E+09,9E+09,9E+09,9E+09,9E+09]];
    CONST robtarget Target_2380:=[[229.198983542,234.781056091,-3],[1,0,0,0],[0,0,0,0],[9E+09,9E+09,9E+09,9E+09,9E+09,9E+09]];
    CONST robtarget Target_1810:=[[118.157953085,231.889203328,-3],[1,0,0,0],[0,0,0,0],[9E+09,9E+09,9E+09,9E+09,9E+09,9E+09]];
    CONST robtarget Target_1720:=[[108.495218386,231.650593675,-3],[1,0,0,0],[0,0,0,0],[9E+09,9E+09,9E+09,9E+09,9E+09,9E+09]];
    CONST robtarget Target_2430:=[[231.736502845,228.588626787,-3],[1,0,0,0],[0,0,0,0],[9E+09,9E+09,9E+09,9E+09,9E+09,9E+09]];
    CONST robtarget Target_2340:=[[224.27087843,226.693925012,-3],[1,0,0,0],[0,0,0,0],[9E+09,9E+09,9E+09,9E+09,9E+09,9E+09]];
    CONST robtarget Target_2550:=[[245.960809109,138.03840632,-3],[1,0,0,0],[0,0,0,0],[9E+09,9E+09,9E+09,9E+09,9E+09,9E+09]];
    CONST robtarget Target_1870:=[[114.097941212,195.477543406,-3],[1,0,0,0],[0,0,0,0],[9E+09,9E+09,9E+09,9E+09,9E+09,9E+09]];
    CONST robtarget Target_2420:=[[234.492086854,230.820271671,-3],[1,0,0,0],[0,0,0,0],[9E+09,9E+09,9E+09,9E+09,9E+09,9E+09]];
    CONST robtarget Target_1680:=[[108.824325808,185.570150163,-3],[1,0,0,0],[0,0,0,0],[9E+09,9E+09,9E+09,9E+09,9E+09,9E+09]];
    CONST robtarget Target_1910:=[[121.949781799,195.938634052,-3],[1,0,0,0],[0,0,0,0],[9E+09,9E+09,9E+09,9E+09,9E+09,9E+09]];
    CONST robtarget Target_2090:=[[163.89131052,175.492184057,-3],[1,0,0,0],[0,0,0,0],[9E+09,9E+09,9E+09,9E+09,9E+09,9E+09]];
    CONST robtarget Target_1740:=[[110.927371266,232.178907073,-3],[1,0,0,0],[0,0,0,0],[9E+09,9E+09,9E+09,9E+09,9E+09,9E+09]];
    CONST robtarget Target_2070:=[[149.13612362,180.924616922,-3],[1,0,0,0],[0,0,0,0],[9E+09,9E+09,9E+09,9E+09,9E+09,9E+09]];
    CONST robtarget Target_2150:=[[193.599222492,215.563562691,-3],[1,0,0,0],[0,0,0,0],[9E+09,9E+09,9E+09,9E+09,9E+09,9E+09]];
    CONST robtarget Target_1670:=[[114.653225127,181.376268279,-3],[1,0,0,0],[0,0,0,0],[9E+09,9E+09,9E+09,9E+09,9E+09,9E+09]];
    CONST robtarget Target_3760:=[[0,0,-20],[1,0,0,0],[0,0,0,0],[9E+09,9E+09,9E+09,9E+09,9E+09,9E+09]];
    CONST robtarget Target_3770:=[[0,297,-20],[1,0,0,0],[0,0,0,0],[9E+09,9E+09,9E+09,9E+09,9E+09,9E+09]];
    CONST robtarget Target_3780:=[[420,297,-20],[1,0,0,0],[0,0,0,0],[9E+09,9E+09,9E+09,9E+09,9E+09,9E+09]];
    CONST robtarget Target_3790:=[[420,0,-20],[1,0,0,0],[0,0,0,0],[9E+09,9E+09,9E+09,9E+09,9E+09,9E+09]];
    CONST robtarget Target_3800:=[[0,0,-20],[1,0,0,0],[0,0,0,0],[9E+09,9E+09,9E+09,9E+09,9E+09,9E+09]];
    !The above varant robot targets are the defined targets to draw the image and the initials
    !The movex variable will be used to translate the coordinates of the targets in refence to the workobject on the x axis
    !The movey variable will be used to translate the coordinates of the targets in refence to the workobject on the y axis
    !Robot targets that draw the outline for number one
    CONST robtarget Target_3810:=[[16.151042905,45.282633581,-3],[1,0,0,0],[0,0,0,0],[9E+09,9E+09,9E+09,9E+09,9E+09,9E+09]];
    CONST robtarget Target_3820:=[[16.23683793,17.577049721,-3],[1,0,0,0],[-1,0,0,0],[9E+09,9E+09,9E+09,9E+09,9E+09,9E+09]];
    CONST robtarget Target_3830:=[[17.639903488,9.237426811,-3],[1,0,0,0],[-1,0,0,0],[9E+09,9E+09,9E+09,9E+09,9E+09,9E+09]];
    CONST robtarget Target_3840:=[[12.87576939,0.139222796,-3],[1,0,0,0],[-1,0,0,0],[9E+09,9E+09,9E+09,9E+09,9E+09,9E+09]];
    CONST robtarget Target_3850:=[[-0.235443238,9.679341092,-3],[1,0,0,0],[-1,0,0,0],[9E+09,9E+09,9E+09,9E+09,9E+09,9E+09]];
    CONST robtarget Target_3860:=[[5.708537709,10.51790976,-3],[1,0,0,0],[-1,0,0,0],[9E+09,9E+09,9E+09,9E+09,9E+09,9E+09]];
    CONST robtarget Target_3870:=[[6.671871038,47.391982572,-3],[1,0,0,0],[-1,0,0,0],[9E+09,9E+09,9E+09,9E+09,9E+09,9E+09]];
    CONST robtarget Target_3880:=[[5.359980624,53.877951817,-3],[1,0,0,0],[-1,0,0,0],[9E+09,9E+09,9E+09,9E+09,9E+09,9E+09]];
    CONST robtarget Target_3890:=[[13.645980545,57.663758501,-3],[1,0,0,0],[-1,0,0,0],[9E+09,9E+09,9E+09,9E+09,9E+09,9E+09]];
    CONST robtarget Target_3900:=[[21.215766786,50.907623325,-3],[1,0,0,0],[-1,0,0,0],[9E+09,9E+09,9E+09,9E+09,9E+09,9E+09]];
    CONST robtarget Target_3910:=[[16.151042905,45.282633581,-3],[1,0,0,0],[-1,0,0,0],[9E+09,9E+09,9E+09,9E+09,9E+09,9E+09]];
    !Robot targets that draw the outline for number two
    CONST robtarget Target_3920:=[[7.881702426,36.119144197,-3],[1,0,0,0],[0,0,0,0],[9E+09,9E+09,9E+09,9E+09,9E+09,9E+09]];
    CONST robtarget Target_3930:=[[1.571425345,44.67698602,-3],[1,0,0,0],[0,0,0,0],[9E+09,9E+09,9E+09,9E+09,9E+09,9E+09]];
    CONST robtarget Target_3940:=[[0.294886856,55.233632159,-3],[1,0,0,0],[0,0,0,0],[9E+09,9E+09,9E+09,9E+09,9E+09,9E+09]];
    CONST robtarget Target_3950:=[[15.913653232,58.440713954,-3],[1,0,0,0],[0,0,0,0],[9E+09,9E+09,9E+09,9E+09,9E+09,9E+09]];
    CONST robtarget Target_3960:=[[28.891932635,58.353249112,-3],[1,0,0,0],[0,0,0,0],[9E+09,9E+09,9E+09,9E+09,9E+09,9E+09]];
    CONST robtarget Target_3970:=[[34.032097662,46.307843859,-3],[1,0,0,0],[0,0,0,0],[9E+09,9E+09,9E+09,9E+09,9E+09,9E+09]];
    CONST robtarget Target_3980:=[[28.17290462,48.356477469,-3],[1,0,0,0],[0,0,0,0],[9E+09,9E+09,9E+09,9E+09,9E+09,9E+09]];
    CONST robtarget Target_3990:=[[10.03552778,48.572348325,-3],[1,0,0,0],[0,0,0,0],[9E+09,9E+09,9E+09,9E+09,9E+09,9E+09]];
    CONST robtarget Target_4000:=[[11.937553493,41.601597978,-3],[1,0,0,0],[0,0,0,0],[9E+09,9E+09,9E+09,9E+09,9E+09,9E+09]];
    CONST robtarget Target_4010:=[[16.49330278,36.7890648,-3],[1,0,0,0],[0,0,0,0],[9E+09,9E+09,9E+09,9E+09,9E+09,9E+09]];
    CONST robtarget Target_4020:=[[22.06071775,32.652738323,-3],[1,0,0,0],[0,0,0,0],[9E+09,9E+09,9E+09,9E+09,9E+09,9E+09]];
    CONST robtarget Target_4030:=[[27.862515872,28.866245564,-3],[1,0,0,0],[0,0,0,0],[9E+09,9E+09,9E+09,9E+09,9E+09,9E+09]];
    CONST robtarget Target_4040:=[[32.551179634,24.228255252,-3],[1,0,0,0],[0,0,0,0],[9E+09,9E+09,9E+09,9E+09,9E+09,9E+09]];
    CONST robtarget Target_4050:=[[33.821892538,17.554132807,-3],[1,0,0,0],[0,0,0,0],[9E+09,9E+09,9E+09,9E+09,9E+09,9E+09]];
    CONST robtarget Target_4060:=[[32.783169698,10.897868553,-3],[1,0,0,0],[0,0,0,0],[9E+09,9E+09,9E+09,9E+09,9E+09,9E+09]];
    CONST robtarget Target_4070:=[[25.544023641,3.255312728,-3],[1,0,0,0],[0,0,0,0],[9E+09,9E+09,9E+09,9E+09,9E+09,9E+09]];
    CONST robtarget Target_4080:=[[3.986848708,7.796787273,-3],[1,0,0,0],[0,0,0,0],[9E+09,9E+09,9E+09,9E+09,9E+09,9E+09]];
    CONST robtarget Target_4090:=[[1.243201105,23.617220142,-3],[1,0,0,0],[0,0,0,0],[9E+09,9E+09,9E+09,9E+09,9E+09,9E+09]];
    CONST robtarget Target_4100:=[[8.95316835,20.654544015,-3],[1,0,0,0],[0,0,0,0],[9E+09,9E+09,9E+09,9E+09,9E+09,9E+09]];
    CONST robtarget Target_4110:=[[10.988772772,13.289311255,-3],[1,0,0,0],[0,0,0,0],[9E+09,9E+09,9E+09,9E+09,9E+09,9E+09]];
    CONST robtarget Target_4120:=[[15.111280691,8.337544795,-3],[1,0,0,0],[0,0,0,0],[9E+09,9E+09,9E+09,9E+09,9E+09,9E+09]];
    CONST robtarget Target_4130:=[[20.521282271,11.790879926,-3],[1,0,0,0],[0,0,0,0],[9E+09,9E+09,9E+09,9E+09,9E+09,9E+09]];
    CONST robtarget Target_4140:=[[23.973453659,18.816230493,-3],[1,0,0,0],[0,0,0,0],[9E+09,9E+09,9E+09,9E+09,9E+09,9E+09]];
    CONST robtarget Target_4150:=[[21.074779646,26.130532237,-3],[1,0,0,0],[0,0,0,0],[9E+09,9E+09,9E+09,9E+09,9E+09,9E+09]];
    CONST robtarget Target_4160:=[[7.881702426,36.119144197,-3],[1,0,0,0],[0,0,0,0],[9E+09,9E+09,9E+09,9E+09,9E+09,9E+09]];
    !Robot targets that draw the outline for number three
    CONST robtarget Target_4170:=[[34.520621698,33.437716008,-3],[1,0,0,0],[0,0,0,0],[9E+09,9E+09,9E+09,9E+09,9E+09,9E+09]];
    CONST robtarget Target_4180:=[[31.592037634,25.979331159,-3],[1,0,0,0],[0,0,0,0],[9E+09,9E+09,9E+09,9E+09,9E+09,9E+09]];
    CONST robtarget Target_4190:=[[25.612746567,21.157477312,-3],[1,0,0,0],[0,0,0,0],[9E+09,9E+09,9E+09,9E+09,9E+09,9E+09]];
    CONST robtarget Target_4200:=[[34.699927182,0.463270809,-3],[1,0,0,0],[0,0,0,0],[9E+09,9E+09,9E+09,9E+09,9E+09,9E+09]];
    CONST robtarget Target_4210:=[[7.818343082,0.396647106,-3],[1,0,0,0],[0,0,0,0],[9E+09,9E+09,9E+09,9E+09,9E+09,9E+09]];
    CONST robtarget Target_4220:=[[2.050615439,10.782787479,-3],[1,0,0,0],[0,0,0,0],[9E+09,9E+09,9E+09,9E+09,9E+09,9E+09]];
    CONST robtarget Target_4230:=[[12.480641301,9.034640293,-3],[1,0,0,0],[0,0,0,0],[9E+09,9E+09,9E+09,9E+09,9E+09,9E+09]];
    CONST robtarget Target_4240:=[[23.232337412,9.283033503,-3],[1,0,0,0],[0,0,0,0],[9E+09,9E+09,9E+09,9E+09,9E+09,9E+09]];
    CONST robtarget Target_4250:=[[9.092214994,27.928019233,-3],[1,0,0,0],[0,0,0,0],[9E+09,9E+09,9E+09,9E+09,9E+09,9E+09]];
    CONST robtarget Target_4260:=[[17.965004549,29.345522284,-3],[1,0,0,0],[0,0,0,0],[9E+09,9E+09,9E+09,9E+09,9E+09,9E+09]];
    CONST robtarget Target_4270:=[[25.277433188,36.212108511,-3],[1,0,0,0],[0,0,0,0],[9E+09,9E+09,9E+09,9E+09,9E+09,9E+09]];
    CONST robtarget Target_4280:=[[25.620291723,43.391200834,-3],[1,0,0,0],[0,0,0,0],[9E+09,9E+09,9E+09,9E+09,9E+09,9E+09]];
    CONST robtarget Target_4290:=[[22.396757747,49.156388346,-3],[1,0,0,0],[0,0,0,0],[9E+09,9E+09,9E+09,9E+09,9E+09,9E+09]];
    CONST robtarget Target_4300:=[[17.057777076,52.455535293,-3],[1,0,0,0],[0,0,0,0],[9E+09,9E+09,9E+09,9E+09,9E+09,9E+09]];
    CONST robtarget Target_4310:=[[10.009672512,47.084506647,-3],[1,0,0,0],[0,0,0,0],[9E+09,9E+09,9E+09,9E+09,9E+09,9E+09]];
    CONST robtarget Target_4320:=[[9.772724831,36.40631401,-3],[1,0,0,0],[0,0,0,0],[9E+09,9E+09,9E+09,9E+09,9E+09,9E+09]];
    CONST robtarget Target_4330:=[[2.938421294,40.207188392,-3],[1,0,0,0],[0,0,0,0],[9E+09,9E+09,9E+09,9E+09,9E+09,9E+09]];
    CONST robtarget Target_4340:=[[0.743684284,48.933949971,-3],[1,0,0,0],[0,0,0,0],[9E+09,9E+09,9E+09,9E+09,9E+09,9E+09]];
    CONST robtarget Target_4350:=[[5.081768353,54.880073404,-3],[1,0,0,0],[0,0,0,0],[9E+09,9E+09,9E+09,9E+09,9E+09,9E+09]];
    CONST robtarget Target_4360:=[[12.765410543,58.26186749,-3],[1,0,0,0],[0,0,0,0],[9E+09,9E+09,9E+09,9E+09,9E+09,9E+09]];
    CONST robtarget Target_4370:=[[20.023231684,57.282904156,-3],[1,0,0,0],[0,0,0,0],[9E+09,9E+09,9E+09,9E+09,9E+09,9E+09]];
    CONST robtarget Target_4380:=[[28.428229984,50.875574385,-3],[1,0,0,0],[0,0,0,0],[9E+09,9E+09,9E+09,9E+09,9E+09,9E+09]];
    CONST robtarget Target_4390:=[[32.41488829,46.190345447,-3],[1,0,0,0],[0,0,0,0],[9E+09,9E+09,9E+09,9E+09,9E+09,9E+09]];
    CONST robtarget Target_4400:=[[34.690272268,40.547802452,-3],[1,0,0,0],[0,0,0,0],[9E+09,9E+09,9E+09,9E+09,9E+09,9E+09]];
    CONST robtarget Target_4410:=[[34.520621698,33.437716008,-3],[1,0,0,0],[0,0,0,0],[9E+09,9E+09,9E+09,9E+09,9E+09,9E+09]];
    !Robot targets that draw the outline for number four
    CONST robtarget Target_4420:=[[20.710461749,0.569865658,-3],[1,0,0,0],[0,0,0,0],[9E+09,9E+09,9E+09,9E+09,9E+09,9E+09]];
    CONST robtarget Target_4430:=[[0.541272032,35.266144788,-3],[1,0,0,0],[0,0,0,0],[9E+09,9E+09,9E+09,9E+09,9E+09,9E+09]];
    CONST robtarget Target_4440:=[[4.036202895,40.829346679,-3],[1,0,0,0],[0,0,0,0],[9E+09,9E+09,9E+09,9E+09,9E+09,9E+09]];
    CONST robtarget Target_4450:=[[16.993483718,40.879712789,-3],[1,0,0,0],[0,0,0,0],[9E+09,9E+09,9E+09,9E+09,9E+09,9E+09]];
    CONST robtarget Target_4460:=[[14.13006043,53.349584785,-3],[1,0,0,0],[0,0,0,0],[9E+09,9E+09,9E+09,9E+09,9E+09,9E+09]];
    CONST robtarget Target_4470:=[[22.113953169,58.603114753,-3],[1,0,0,0],[0,0,0,0],[9E+09,9E+09,9E+09,9E+09,9E+09,9E+09]];
    CONST robtarget Target_4480:=[[29.140950033,51.231617827,-3],[1,0,0,0],[0,0,0,0],[9E+09,9E+09,9E+09,9E+09,9E+09,9E+09]];
    CONST robtarget Target_4490:=[[24.807750744,45.809691511,-3],[1,0,0,0],[0,0,0,0],[9E+09,9E+09,9E+09,9E+09,9E+09,9E+09]];
    CONST robtarget Target_4500:=[[30.059232219,40.113789707,-3],[1,0,0,0],[0,0,0,0],[9E+09,9E+09,9E+09,9E+09,9E+09,9E+09]];
    CONST robtarget Target_4510:=[[35.946122293,35.021043979,-3],[1,0,0,0],[0,0,0,0],[9E+09,9E+09,9E+09,9E+09,9E+09,9E+09]];
    CONST robtarget Target_4520:=[[25.697133224,32.221775045,-3],[1,0,0,0],[0,0,0,0],[9E+09,9E+09,9E+09,9E+09,9E+09,9E+09]];
    CONST robtarget Target_4530:=[[25.124293518,20.456615051,-3],[1,0,0,0],[0,0,0,0],[9E+09,9E+09,9E+09,9E+09,9E+09,9E+09]];
    CONST robtarget Target_4540:=[[24.902097043,10.189942803,-3],[1,0,0,0],[0,0,0,0],[9E+09,9E+09,9E+09,9E+09,9E+09,9E+09]];
    CONST robtarget Target_4550:=[[22.502567351,0.574308873,-3],[1,0,0,0],[0,0,0,0],[9E+09,9E+09,9E+09,9E+09,9E+09,9E+09]];
    CONST robtarget Target_4560:=[[20.710461749,0.569865658,-3],[1,0,0,0],[0,0,0,0],[9E+09,9E+09,9E+09,9E+09,9E+09,9E+09]];
    CONST robtarget Target_4570:=[[20.71,0.57,-23],[1,0,0,0],[0,0,0,0],[9E+09,9E+09,9E+09,9E+09,9E+09,9E+09]];
    CONST robtarget Target_4571:=[[15.995,31.768,-23],[1,0,0,0],[0,0,0,0],[9E+09,9E+09,9E+09,9E+09,9E+09,9E+09]];
    CONST robtarget Target_4580:=[[15.994847275,31.767946317,-3],[1,0,0,0],[0,0,0,0],[9E+09,9E+09,9E+09,9E+09,9E+09,9E+09]];
    CONST robtarget Target_4590:=[[8.052701519,31.74826272,-3],[1,0,0,0],[0,0,0,0],[9E+09,9E+09,9E+09,9E+09,9E+09,9E+09]];
    CONST robtarget Target_4600:=[[15.165368404,18.039347459,-3],[1,0,0,0],[0,0,0,0],[9E+09,9E+09,9E+09,9E+09,9E+09,9E+09]];
    CONST robtarget Target_4610:=[[15.994847275,31.767946317,-3],[1,0,0,0],[0,0,0,0],[9E+09,9E+09,9E+09,9E+09,9E+09,9E+09]];
    !Robot targets that draw the outline for number five
    CONST robtarget Target_4620:=[[15.577577146,0.700891672,-3],[1,0,0,0],[0,0,0,0],[9E+09,9E+09,9E+09,9E+09,9E+09,9E+09]];
    CONST robtarget Target_4630:=[[3.381822569,30.438211842,-3],[1,0,0,0],[0,0,0,0],[9E+09,9E+09,9E+09,9E+09,9E+09,9E+09]];
    CONST robtarget Target_4640:=[[16.397500703,29.526893677,-3],[1,0,0,0],[0,0,0,0],[9E+09,9E+09,9E+09,9E+09,9E+09,9E+09]];
    CONST robtarget Target_4650:=[[22.587269316,33.671957362,-3],[1,0,0,0],[0,0,0,0],[9E+09,9E+09,9E+09,9E+09,9E+09,9E+09]];
    CONST robtarget Target_4660:=[[25.474580048,41.336688627,-3],[1,0,0,0],[0,0,0,0],[9E+09,9E+09,9E+09,9E+09,9E+09,9E+09]];
    CONST robtarget Target_4670:=[[23.263122198,49.204078015,-3],[1,0,0,0],[0,0,0,0],[9E+09,9E+09,9E+09,9E+09,9E+09,9E+09]];
    CONST robtarget Target_4680:=[[18.238366809,53.248193939,-3],[1,0,0,0],[0,0,0,0],[9E+09,9E+09,9E+09,9E+09,9E+09,9E+09]];
    CONST robtarget Target_4690:=[[12.038192106,48.431906309,-3],[1,0,0,0],[0,0,0,0],[9E+09,9E+09,9E+09,9E+09,9E+09,9E+09]];
    CONST robtarget Target_4700:=[[10.44880667,40.204253873,-3],[1,0,0,0],[0,0,0,0],[9E+09,9E+09,9E+09,9E+09,9E+09,9E+09]];
    CONST robtarget Target_4710:=[[1.530450653,44.445833761,-3],[1,0,0,0],[0,0,0,0],[9E+09,9E+09,9E+09,9E+09,9E+09,9E+09]];
    CONST robtarget Target_4720:=[[2.141702003,52.450696359,-3],[1,0,0,0],[0,0,0,0],[9E+09,9E+09,9E+09,9E+09,9E+09,9E+09]];
    CONST robtarget Target_4730:=[[9.352457121,58.024560551,-3],[1,0,0,0],[0,0,0,0],[9E+09,9E+09,9E+09,9E+09,9E+09,9E+09]];
    CONST robtarget Target_4740:=[[18.369252239,58.591458604,-3],[1,0,0,0],[0,0,0,0],[9E+09,9E+09,9E+09,9E+09,9E+09,9E+09]];
    CONST robtarget Target_4750:=[[27.605195591,52.757328981,-3],[1,0,0,0],[0,0,0,0],[9E+09,9E+09,9E+09,9E+09,9E+09,9E+09]];
    CONST robtarget Target_4760:=[[31.307603234,46.897822914,-3],[1,0,0,0],[0,0,0,0],[9E+09,9E+09,9E+09,9E+09,9E+09,9E+09]];
    CONST robtarget Target_4770:=[[33.562281366,40.305584434,-3],[1,0,0,0],[0,0,0,0],[9E+09,9E+09,9E+09,9E+09,9E+09,9E+09]];
    CONST robtarget Target_4780:=[[33.880004965,34.062533015,-3],[1,0,0,0],[0,0,0,0],[9E+09,9E+09,9E+09,9E+09,9E+09,9E+09]];
    CONST robtarget Target_4790:=[[29.292032597,24.630522538,-3],[1,0,0,0],[0,0,0,0],[9E+09,9E+09,9E+09,9E+09,9E+09,9E+09]];
    CONST robtarget Target_4800:=[[19.692642123,20.175173927,-3],[1,0,0,0],[0,0,0,0],[9E+09,9E+09,9E+09,9E+09,9E+09,9E+09]];
    CONST robtarget Target_4810:=[[13.530279259,19.631749741,-3],[1,0,0,0],[0,0,0,0],[9E+09,9E+09,9E+09,9E+09,9E+09,9E+09]];
    CONST robtarget Target_4820:=[[15.713993933,12.443389191,-3],[1,0,0,0],[0,0,0,0],[9E+09,9E+09,9E+09,9E+09,9E+09,9E+09]];
    CONST robtarget Target_4830:=[[27.058831577,11.342264171,-3],[1,0,0,0],[0,0,0,0],[9E+09,9E+09,9E+09,9E+09,9E+09,9E+09]];
    CONST robtarget Target_4840:=[[35.19592993,4.530940095,-3],[1,0,0,0],[0,0,0,0],[9E+09,9E+09,9E+09,9E+09,9E+09,9E+09]];
    CONST robtarget Target_4850:=[[15.577577146,0.700891672,-3],[1,0,0,0],[0,0,0,0],[9E+09,9E+09,9E+09,9E+09,9E+09,9E+09]];
    !Robot targets that draw the outline for number six
    CONST robtarget Target_4860:=[[0.175773411,12.655991979,-3],[1,0,0,0],[0,0,0,0],[9E+09,9E+09,9E+09,9E+09,9E+09,9E+09]];
    CONST robtarget Target_4870:=[[0.095826313,44.913892901,-3],[1,0,0,0],[0,0,0,0],[9E+09,9E+09,9E+09,9E+09,9E+09,9E+09]];
    CONST robtarget Target_4880:=[[5.352343091,52.864914091,-3],[1,0,0,0],[0,0,0,0],[9E+09,9E+09,9E+09,9E+09,9E+09,9E+09]];
    CONST robtarget Target_4890:=[[13.489402197,57.804804695,-3],[1,0,0,0],[0,0,0,0],[9E+09,9E+09,9E+09,9E+09,9E+09,9E+09]];
    CONST robtarget Target_4900:=[[22.038084304,55.709597939,-3],[1,0,0,0],[0,0,0,0],[9E+09,9E+09,9E+09,9E+09,9E+09,9E+09]];
    CONST robtarget Target_4910:=[[26.724472287,51.458953761,-3],[1,0,0,0],[0,0,0,0],[9E+09,9E+09,9E+09,9E+09,9E+09,9E+09]];
    CONST robtarget Target_4920:=[[33.353883011,46.317068519,-3],[1,0,0,0],[0,0,0,0],[9E+09,9E+09,9E+09,9E+09,9E+09,9E+09]];
    CONST robtarget Target_4930:=[[35.125636077,39.426715999,-3],[1,0,0,0],[0,0,0,0],[9E+09,9E+09,9E+09,9E+09,9E+09,9E+09]];
    CONST robtarget Target_4940:=[[31.654530325,29.413974627,-3],[1,0,0,0],[0,0,0,0],[9E+09,9E+09,9E+09,9E+09,9E+09,9E+09]];
    CONST robtarget Target_4950:=[[24.591760186,23.125142128,-3],[1,0,0,0],[0,0,0,0],[9E+09,9E+09,9E+09,9E+09,9E+09,9E+09]];
    CONST robtarget Target_4960:=[[10.703707271,30.026122869,-3],[1,0,0,0],[0,0,0,0],[9E+09,9E+09,9E+09,9E+09,9E+09,9E+09]];
    CONST robtarget Target_4970:=[[10.621924903,21.9721123,-3],[1,0,0,0],[0,0,0,0],[9E+09,9E+09,9E+09,9E+09,9E+09,9E+09]];
    CONST robtarget Target_4980:=[[10.892215228,14.789387627,-3],[1,0,0,0],[0,0,0,0],[9E+09,9E+09,9E+09,9E+09,9E+09,9E+09]];
    CONST robtarget Target_4990:=[[14.193986227,9.29945116,-3],[1,0,0,0],[0,0,0,0],[9E+09,9E+09,9E+09,9E+09,9E+09,9E+09]];
    CONST robtarget Target_5000:=[[23.502552544,14.033989334,-3],[1,0,0,0],[0,0,0,0],[9E+09,9E+09,9E+09,9E+09,9E+09,9E+09]];
    CONST robtarget Target_5010:=[[33.282953434,11.932369411,-3],[1,0,0,0],[0,0,0,0],[9E+09,9E+09,9E+09,9E+09,9E+09,9E+09]];
    CONST robtarget Target_5020:=[[27.560727715,4.941597888,-3],[1,0,0,0],[0,0,0,0],[9E+09,9E+09,9E+09,9E+09,9E+09,9E+09]];
    CONST robtarget Target_5030:=[[22.162331593,1.111887678,-3],[1,0,0,0],[0,0,0,0],[9E+09,9E+09,9E+09,9E+09,9E+09,9E+09]];
    CONST robtarget Target_5040:=[[15.540941071,0.738901102,-3],[1,0,0,0],[0,0,0,0],[9E+09,9E+09,9E+09,9E+09,9E+09,9E+09]];
    CONST robtarget Target_5050:=[[6.59636995,5.077513585,-3],[1,0,0,0],[0,0,0,0],[9E+09,9E+09,9E+09,9E+09,9E+09,9E+09]];
    CONST robtarget Target_5060:=[[0.175773411,12.655991979,-3],[1,0,0,0],[0,0,0,0],[9E+09,9E+09,9E+09,9E+09,9E+09,9E+09]];
    CONST robtarget Target_5070:=[[0.176,12.656,-23],[1,0,0,0],[0,0,0,0],[9E+09,9E+09,9E+09,9E+09,9E+09,9E+09]];
    CONST robtarget Target_5071:=[[16.872,49.459,-23],[1,0,0,0],[0,0,0,0],[9E+09,9E+09,9E+09,9E+09,9E+09,9E+09]];
    CONST robtarget Target_5080:=[[16.871923709,49.459210649,-3],[1,0,0,0],[0,0,0,0],[9E+09,9E+09,9E+09,9E+09,9E+09,9E+09]];
    CONST robtarget Target_5090:=[[10.430228431,41.142643589,-3],[1,0,0,0],[0,0,0,0],[9E+09,9E+09,9E+09,9E+09,9E+09,9E+09]];
    CONST robtarget Target_5100:=[[15.531115859,31.907468394,-3],[1,0,0,0],[0,0,0,0],[9E+09,9E+09,9E+09,9E+09,9E+09,9E+09]];
    CONST robtarget Target_5110:=[[23.502680148,36.980622333,-3],[1,0,0,0],[0,0,0,0],[9E+09,9E+09,9E+09,9E+09,9E+09,9E+09]];
    CONST robtarget Target_5120:=[[24.096037987,42.95982733,-3],[1,0,0,0],[0,0,0,0],[9E+09,9E+09,9E+09,9E+09,9E+09,9E+09]];
    CONST robtarget Target_5130:=[[16.871923709,49.459210649,-3],[1,0,0,0],[0,0,0,0],[9E+09,9E+09,9E+09,9E+09,9E+09,9E+09]];
    !Robot targets that draw the outline for number seven
    CONST robtarget Target_5140:=[[1.161126116,17.449711773,-3],[1,0,0,0],[0,0,0,0],[9E+09,9E+09,9E+09,9E+09,9E+09,9E+09]];
    CONST robtarget Target_5150:=[[6.907064598,13.739199525,-3],[1,0,0,0],[0,0,0,0],[9E+09,9E+09,9E+09,9E+09,9E+09,9E+09]];
    CONST robtarget Target_5160:=[[12.953826529,12.454981073,-3],[1,0,0,0],[0,0,0,0],[9E+09,9E+09,9E+09,9E+09,9E+09,9E+09]];
    CONST robtarget Target_5170:=[[25.401264788,12.756929769,-3],[1,0,0,0],[0,0,0,0],[9E+09,9E+09,9E+09,9E+09,9E+09,9E+09]];
    CONST robtarget Target_5180:=[[13.126505085,34.940519254,-3],[1,0,0,0],[0,0,0,0],[9E+09,9E+09,9E+09,9E+09,9E+09,9E+09]];
    CONST robtarget Target_5190:=[[10.158608628,41.39549339,-3],[1,0,0,0],[0,0,0,0],[9E+09,9E+09,9E+09,9E+09,9E+09,9E+09]];
    CONST robtarget Target_5200:=[[7.907607757,48.140766941,-3],[1,0,0,0],[0,0,0,0],[9E+09,9E+09,9E+09,9E+09,9E+09,9E+09]];
    CONST robtarget Target_5210:=[[8.287282874,54.607372051,-3],[1,0,0,0],[0,0,0,0],[9E+09,9E+09,9E+09,9E+09,9E+09,9E+09]];
    CONST robtarget Target_5220:=[[12.252476768,59.229851723,-3],[1,0,0,0],[0,0,0,0],[9E+09,9E+09,9E+09,9E+09,9E+09,9E+09]];
    CONST robtarget Target_5230:=[[22.015880386,50.633152169,-3],[1,0,0,0],[0,0,0,0],[9E+09,9E+09,9E+09,9E+09,9E+09,9E+09]];
    CONST robtarget Target_5240:=[[19.080506535,45.13961202,-3],[1,0,0,0],[0,0,0,0],[9E+09,9E+09,9E+09,9E+09,9E+09,9E+09]];
    CONST robtarget Target_5250:=[[19.549471726,38.686108186,-3],[1,0,0,0],[0,0,0,0],[9E+09,9E+09,9E+09,9E+09,9E+09,9E+09]];
    CONST robtarget Target_5260:=[[21.27523326,32.453933068,-3],[1,0,0,0],[0,0,0,0],[9E+09,9E+09,9E+09,9E+09,9E+09,9E+09]];
    CONST robtarget Target_5270:=[[23.788389006,26.533377018,-3],[1,0,0,0],[0,0,0,0],[9E+09,9E+09,9E+09,9E+09,9E+09,9E+09]];
    CONST robtarget Target_5280:=[[30.159183996,15.351372753,-3],[1,0,0,0],[0,0,0,0],[9E+09,9E+09,9E+09,9E+09,9E+09,9E+09]];
    CONST robtarget Target_5290:=[[36.813771449,4.255343737,-3],[1,0,0,0],[0,0,0,0],[9E+09,9E+09,9E+09,9E+09,9E+09,9E+09]];
    CONST robtarget Target_5300:=[[23.723351712,4.210987549,-3],[1,0,0,0],[0,0,0,0],[9E+09,9E+09,9E+09,9E+09,9E+09,9E+09]];
    CONST robtarget Target_5310:=[[17.636911215,4.001175032,-3],[1,0,0,0],[0,0,0,0],[9E+09,9E+09,9E+09,9E+09,9E+09,9E+09]];
    CONST robtarget Target_5320:=[[11.673368623,2.132673866,-3],[1,0,0,0],[0,0,0,0],[9E+09,9E+09,9E+09,9E+09,9E+09,9E+09]];
    CONST robtarget Target_5330:=[[-0.011776561,15.617409476,-3],[1,0,0,0],[0,0,0,0],[9E+09,9E+09,9E+09,9E+09,9E+09,9E+09]];
    CONST robtarget Target_5340:=[[1.161126116,17.449711773,-3],[1,0,0,0],[0,0,0,0],[9E+09,9E+09,9E+09,9E+09,9E+09,9E+09]];
    !Robot targets that draw the outline for number eight
    CONST robtarget Target_5350:=[[18.880343282,1.386145652,-3],[1,0,0,0],[0,0,0,0],[9E+09,9E+09,9E+09,9E+09,9E+09,9E+09]];
    CONST robtarget Target_5360:=[[9.115582726,9.915230022,-3],[1,0,0,0],[0,0,0,0],[9E+09,9E+09,9E+09,9E+09,9E+09,9E+09]];
    CONST robtarget Target_5370:=[[5.158678676,14.858900528,-3],[1,0,0,0],[0,0,0,0],[9E+09,9E+09,9E+09,9E+09,9E+09,9E+09]];
    CONST robtarget Target_5380:=[[5.208573592,25.997381079,-3],[1,0,0,0],[0,0,0,0],[9E+09,9E+09,9E+09,9E+09,9E+09,9E+09]];
    CONST robtarget Target_5390:=[[10.852648949,30.693168127,-3],[1,0,0,0],[0,0,0,0],[9E+09,9E+09,9E+09,9E+09,9E+09,9E+09]];
    CONST robtarget Target_5400:=[[6.327105166,34.757215371,-3],[1,0,0,0],[0,0,0,0],[9E+09,9E+09,9E+09,9E+09,9E+09,9E+09]];
    CONST robtarget Target_5410:=[[1.999328759,39.065287555,-3],[1,0,0,0],[0,0,0,0],[9E+09,9E+09,9E+09,9E+09,9E+09,9E+09]];
    CONST robtarget Target_5420:=[[1.986853359,47.709415615,-3],[1,0,0,0],[0,0,0,0],[9E+09,9E+09,9E+09,9E+09,9E+09,9E+09]];
    CONST robtarget Target_5430:=[[6.376902652,51.914046986,-3],[1,0,0,0],[0,0,0,0],[9E+09,9E+09,9E+09,9E+09,9E+09,9E+09]];
    CONST robtarget Target_5440:=[[12.277774107,55.364064766,-3],[1,0,0,0],[0,0,0,0],[9E+09,9E+09,9E+09,9E+09,9E+09,9E+09]];
    CONST robtarget Target_5450:=[[18.416888421,58.475461963,-3],[1,0,0,0],[0,0,0,0],[9E+09,9E+09,9E+09,9E+09,9E+09,9E+09]];
    CONST robtarget Target_5460:=[[26.463803828,51.198291716,-3],[1,0,0,0],[0,0,0,0],[9E+09,9E+09,9E+09,9E+09,9E+09,9E+09]];
    CONST robtarget Target_5470:=[[35.710332413,43.493976727,-3],[1,0,0,0],[0,0,0,0],[9E+09,9E+09,9E+09,9E+09,9E+09,9E+09]];
    CONST robtarget Target_5480:=[[38.336065575,37.353723701,-3],[1,0,0,0],[0,0,0,0],[9E+09,9E+09,9E+09,9E+09,9E+09,9E+09]];
    CONST robtarget Target_5490:=[[34.603904904,31.687974352,-3],[1,0,0,0],[0,0,0,0],[9E+09,9E+09,9E+09,9E+09,9E+09,9E+09]];
    CONST robtarget Target_5500:=[[34.954203208,22.534714628,-3],[1,0,0,0],[0,0,0,0],[9E+09,9E+09,9E+09,9E+09,9E+09,9E+09]];
    CONST robtarget Target_5510:=[[37.829730689,12.712769298,-3],[1,0,0,0],[0,0,0,0],[9E+09,9E+09,9E+09,9E+09,9E+09,9E+09]];
    CONST robtarget Target_5520:=[[31.218819854,4.990266122,-3],[1,0,0,0],[0,0,0,0],[9E+09,9E+09,9E+09,9E+09,9E+09,9E+09]];
    CONST robtarget Target_5530:=[[22.33505193,0.813396444,-3],[1,0,0,0],[0,0,0,0],[9E+09,9E+09,9E+09,9E+09,9E+09,9E+09]];
    CONST robtarget Target_5540:=[[18.880343282,1.386145652,-3],[1,0,0,0],[0,0,0,0],[9E+09,9E+09,9E+09,9E+09,9E+09,9E+09]];
    CONST robtarget Target_5540_2:=[[18.88,1.386,-23],[1,0,0,0],[0,0,0,0],[9E+09,9E+09,9E+09,9E+09,9E+09,9E+09]];
    CONST robtarget Target_5610:=[[17.442109817,9.51056124,-3],[1,0,0,0],[0,0,0,0],[9E+09,9E+09,9E+09,9E+09,9E+09,9E+09]];
    CONST robtarget Target_5550:=[[17.442109817,9.51056124,-3],[1,0,0,0],[0,0,0,0],[9E+09,9E+09,9E+09,9E+09,9E+09,9E+09]];
    CONST robtarget Target_5560:=[[23.516133595,11.466033191,-3],[1,0,0,0],[0,0,0,0],[9E+09,9E+09,9E+09,9E+09,9E+09,9E+09]];
    CONST robtarget Target_5570:=[[29.134760604,18.967181282,-3],[1,0,0,0],[0,0,0,0],[9E+09,9E+09,9E+09,9E+09,9E+09,9E+09]];
    CONST robtarget Target_5580:=[[24.576313909,25.000496807,-3],[1,0,0,0],[0,0,0,0],[9E+09,9E+09,9E+09,9E+09,9E+09,9E+09]];
    CONST robtarget Target_5590:=[[15.787410503,21.473452726,-3],[1,0,0,0],[0,0,0,0],[9E+09,9E+09,9E+09,9E+09,9E+09,9E+09]];
    CONST robtarget Target_5600:=[[12.788989878,15.580955105,-3],[1,0,0,0],[0,0,0,0],[9E+09,9E+09,9E+09,9E+09,9E+09,9E+09]];
    CONST robtarget Target_5610_2:=[[17.442,9.511,-23],[1,0,0,0],[0,0,0,0],[9E+09,9E+09,9E+09,9E+09,9E+09,9E+09]];
    CONST robtarget Target_5620:=[[21.450682213,48.953925224,-3],[1,0,0,0],[0,0,0,0],[9E+09,9E+09,9E+09,9E+09,9E+09,9E+09]];
    CONST robtarget Target_5630:=[[16.056172273,44.36292767,-3],[1,0,0,0],[0,0,0,0],[9E+09,9E+09,9E+09,9E+09,9E+09,9E+09]];
    CONST robtarget Target_5640:=[[11.070257525,39.754689626,-3],[1,0,0,0],[0,0,0,0],[9E+09,9E+09,9E+09,9E+09,9E+09,9E+09]];
    CONST robtarget Target_5650:=[[15.590169984,34.400334749,-3],[1,0,0,0],[0,0,0,0],[9E+09,9E+09,9E+09,9E+09,9E+09,9E+09]];
    CONST robtarget Target_5660:=[[22.659943048,36.648427695,-3],[1,0,0,0],[0,0,0,0],[9E+09,9E+09,9E+09,9E+09,9E+09,9E+09]];
    CONST robtarget Target_5670:=[[29.195196496,41.399771231,-3],[1,0,0,0],[0,0,0,0],[9E+09,9E+09,9E+09,9E+09,9E+09,9E+09]];
    CONST robtarget Target_5680:=[[21.450682213,48.953925224,-3],[1,0,0,0],[0,0,0,0],[9E+09,9E+09,9E+09,9E+09,9E+09,9E+09]];
    !Robot targets that draw the outline for number nine
    CONST robtarget Target_5690:=[[13.241409665,1.822069964,-3],[1,0,0,0],[0,0,0,0],[9E+09,9E+09,9E+09,9E+09,9E+09,9E+09]];
    CONST robtarget Target_5700:=[[6.803893377,6.386082993,-3],[1,0,0,0],[0,0,0,0],[9E+09,9E+09,9E+09,9E+09,9E+09,9E+09]];
    CONST robtarget Target_5710:=[[2.66437496,12.310655694,-3],[1,0,0,0],[0,0,0,0],[9E+09,9E+09,9E+09,9E+09,9E+09,9E+09]];
    CONST robtarget Target_5720:=[[0.938639364,19.340063829,-3],[1,0,0,0],[0,0,0,0],[9E+09,9E+09,9E+09,9E+09,9E+09,9E+09]];
    CONST robtarget Target_5730:=[[1.742471539,27.218583159,-3],[1,0,0,0],[0,0,0,0],[9E+09,9E+09,9E+09,9E+09,9E+09,9E+09]];
    CONST robtarget Target_5740:=[[9.388997937,35.266842952,-3],[1,0,0,0],[0,0,0,0],[9E+09,9E+09,9E+09,9E+09,9E+09,9E+09]];
    CONST robtarget Target_5750:=[[20.302452005,34.392316999,-3],[1,0,0,0],[0,0,0,0],[9E+09,9E+09,9E+09,9E+09,9E+09,9E+09]];
    CONST robtarget Target_5760:=[[22.253270414,42.581930294,-3],[1,0,0,0],[0,0,0,0],[9E+09,9E+09,9E+09,9E+09,9E+09,9E+09]];
    CONST robtarget Target_5770:=[[13.667789926,50.421820301,-3],[1,0,0,0],[0,0,0,0],[9E+09,9E+09,9E+09,9E+09,9E+09,9E+09]];
    CONST robtarget Target_5780:=[[9.576140268,40.907891327,-3],[1,0,0,0],[0,0,0,0],[9E+09,9E+09,9E+09,9E+09,9E+09,9E+09]];
    CONST robtarget Target_5790:=[[1.762741471,44.350735745,-3],[1,0,0,0],[0,0,0,0],[9E+09,9E+09,9E+09,9E+09,9E+09,9E+09]];
    CONST robtarget Target_5800:=[[1.529179969,52.175293766,-3],[1,0,0,0],[0,0,0,0],[9E+09,9E+09,9E+09,9E+09,9E+09,9E+09]];
    CONST robtarget Target_5810:=[[6.939405015,55.802236284,-3],[1,0,0,0],[0,0,0,0],[9E+09,9E+09,9E+09,9E+09,9E+09,9E+09]];
    CONST robtarget Target_5820:=[[16.660320643,58.61981089,-3],[1,0,0,0],[0,0,0,0],[9E+09,9E+09,9E+09,9E+09,9E+09,9E+09]];
    CONST robtarget Target_5830:=[[33.188791099,45.286253917,-3],[1,0,0,0],[0,0,0,0],[9E+09,9E+09,9E+09,9E+09,9E+09,9E+09]];
    CONST robtarget Target_5840:=[[34.752223793,14.913374701,-3],[1,0,0,0],[0,0,0,0],[9E+09,9E+09,9E+09,9E+09,9E+09,9E+09]];
    CONST robtarget Target_5850:=[[32.746117885,7.609630004,-3],[1,0,0,0],[0,0,0,0],[9E+09,9E+09,9E+09,9E+09,9E+09,9E+09]];
    CONST robtarget Target_5860:=[[27.633867916,2.469512313,-3],[1,0,0,0],[0,0,0,0],[9E+09,9E+09,9E+09,9E+09,9E+09,9E+09]];
    CONST robtarget Target_5870:=[[20.703092353,0.278499632,-3],[1,0,0,0],[0,0,0,0],[9E+09,9E+09,9E+09,9E+09,9E+09,9E+09]];
    CONST robtarget Target_5880:=[[13.241409665,1.822069964,-3],[1,0,0,0],[0,0,0,0],[9E+09,9E+09,9E+09,9E+09,9E+09,9E+09]];
    CONST robtarget Target_5880_2:=[[13.241,1.822,-23],[1,0,0,0],[0,0,0,0],[9E+09,9E+09,9E+09,9E+09,9E+09,9E+09]];
    CONST robtarget Target_5890:=[[12.894604575,14.707538234,-3],[1,0,0,0],[0,0,0,0],[9E+09,9E+09,9E+09,9E+09,9E+09,9E+09]];
    CONST robtarget Target_5900:=[[18.454763865,8.663996491,-3],[1,0,0,0],[0,0,0,0],[9E+09,9E+09,9E+09,9E+09,9E+09,9E+09]];
    CONST robtarget Target_5910:=[[24.84806073,15.932033095,-3],[1,0,0,0],[0,0,0,0],[9E+09,9E+09,9E+09,9E+09,9E+09,9E+09]];
    CONST robtarget Target_5920:=[[24.194682569,23.634692815,-3],[1,0,0,0],[0,0,0,0],[9E+09,9E+09,9E+09,9E+09,9E+09,9E+09]];
    CONST robtarget Target_5930:=[[19.107180515,28.688646578,-3],[1,0,0,0],[0,0,0,0],[9E+09,9E+09,9E+09,9E+09,9E+09,9E+09]];
    CONST robtarget Target_5940:=[[13.584065215,26.337903975,-3],[1,0,0,0],[0,0,0,0],[9E+09,9E+09,9E+09,9E+09,9E+09,9E+09]];
    CONST robtarget Target_5950:=[[12.436606626,18.938803184,-3],[1,0,0,0],[0,0,0,0],[9E+09,9E+09,9E+09,9E+09,9E+09,9E+09]];
    CONST robtarget Target_5960:=[[12.894604575,14.707538234,-3],[1,0,0,0],[0,0,0,0],[9E+09,9E+09,9E+09,9E+09,9E+09,9E+09]];
    !Robot targets that draw the outline for number zero
    CONST robtarget Target_5970:=[[-0.208072129,14.064489024,-3],[1,0,0,0],[0,0,0,0],[9E+09,9E+09,9E+09,9E+09,9E+09,9E+09]];
    CONST robtarget Target_5980:=[[0.238206781,44.473317866,-3],[1,0,0,0],[-1,0,0,0],[9E+09,9E+09,9E+09,9E+09,9E+09,9E+09]];
    CONST robtarget Target_5990:=[[9.645521629,50.69637459,-3],[1,0,0,0],[-1,0,0,0],[9E+09,9E+09,9E+09,9E+09,9E+09,9E+09]];
    CONST robtarget Target_6000:=[[15.258688414,55.216918654,-3],[1,0,0,0],[-1,0,0,0],[9E+09,9E+09,9E+09,9E+09,9E+09,9E+09]];
    CONST robtarget Target_6010:=[[20.640016881,58.775263581,-3],[1,0,0,0],[-1,0,0,0],[9E+09,9E+09,9E+09,9E+09,9E+09,9E+09]];
    CONST robtarget Target_6020:=[[29.835994744,51.215399122,-3],[1,0,0,0],[-1,0,0,0],[9E+09,9E+09,9E+09,9E+09,9E+09,9E+09]];
    CONST robtarget Target_6030:=[[34.422966873,41.172472481,-3],[1,0,0,0],[-1,0,0,0],[9E+09,9E+09,9E+09,9E+09,9E+09,9E+09]];
    CONST robtarget Target_6040:=[[34.123325729,30.428074706,-3],[1,0,0,0],[-1,0,0,0],[9E+09,9E+09,9E+09,9E+09,9E+09,9E+09]];
    CONST robtarget Target_6050:=[[34.420577684,19.694016205,-3],[1,0,0,0],[-1,0,0,0],[9E+09,9E+09,9E+09,9E+09,9E+09,9E+09]];
    CONST robtarget Target_6060:=[[33.192150654,11.301900797,-3],[1,0,0,0],[-1,0,0,0],[9E+09,9E+09,9E+09,9E+09,9E+09,9E+09]];
    CONST robtarget Target_6070:=[[23.520993793,4.360430914,-3],[1,0,0,0],[-1,0,0,0],[9E+09,9E+09,9E+09,9E+09,9E+09,9E+09]];
    CONST robtarget Target_6080:=[[17.927467446,0.731052411,-3],[1,0,0,0],[-1,0,0,0],[9E+09,9E+09,9E+09,9E+09,9E+09,9E+09]];
    CONST robtarget Target_6090:=[[7.212781677,5.188566065,-3],[1,0,0,0],[-1,0,0,0],[9E+09,9E+09,9E+09,9E+09,9E+09,9E+09]];
    CONST robtarget Target_6100:=[[1.976022879,9.698480519,-3],[1,0,0,0],[-1,0,0,0],[9E+09,9E+09,9E+09,9E+09,9E+09,9E+09]];
    CONST robtarget Target_6110:=[[-0.208072129,14.064489024,-3],[1,0,0,0],[-1,0,0,0],[9E+09,9E+09,9E+09,9E+09,9E+09,9E+09]];
    CONST robtarget Target_6110_2:=[[-0.208,14.064,-23],[1,0,0,0],[-1,0,0,0],[9E+09,9E+09,9E+09,9E+09,9E+09,9E+09]];
    CONST robtarget Target_6200:=[[11.619404059,27.387038013,-3],[1,0,0,0],[-1,0,0,0],[9E+09,9E+09,9E+09,9E+09,9E+09,9E+09]];
    CONST robtarget Target_6120:=[[11.619404059,27.387038013,-3],[1,0,0,0],[-1,0,0,0],[9E+09,9E+09,9E+09,9E+09,9E+09,9E+09]];
    CONST robtarget Target_6130:=[[11.704708697,14.449963254,-3],[1,0,0,0],[-1,0,0,0],[9E+09,9E+09,9E+09,9E+09,9E+09,9E+09]];
    CONST robtarget Target_6140:=[[15.796492768,9.637786231,-3],[1,0,0,0],[-1,0,0,0],[9E+09,9E+09,9E+09,9E+09,9E+09,9E+09]];
    CONST robtarget Target_6150:=[[22.803826625,14.845127374,-3],[1,0,0,0],[-1,0,0,0],[9E+09,9E+09,9E+09,9E+09,9E+09,9E+09]];
    CONST robtarget Target_6160:=[[24.118672366,45.158373362,-3],[1,0,0,0],[-1,0,0,0],[9E+09,9E+09,9E+09,9E+09,9E+09,9E+09]];
    CONST robtarget Target_6170:=[[17.634665749,48.501072917,-3],[1,0,0,0],[-1,0,0,0],[9E+09,9E+09,9E+09,9E+09,9E+09,9E+09]];
    CONST robtarget Target_6180:=[[12.796185416,44.123451337,-3],[1,0,0,0],[-1,0,0,0],[9E+09,9E+09,9E+09,9E+09,9E+09,9E+09]];
    CONST robtarget Target_6190:=[[11.519803934,37.64042127,-3],[1,0,0,0],[-1,0,0,0],[9E+09,9E+09,9E+09,9E+09,9E+09,9E+09]];
    CONST robtarget Target_1640_2:=[[116.864,164.593,-23],[1,0,0,0],[0,0,0,0],[9E+09,9E+09,9E+09,9E+09,9E+09,9E+09]];
    CONST robtarget Target_1641:=[[116.864395565,164.59256718,-3],[1,0,0,0],[0,0,0,0],[9E+09,9E+09,9E+09,9E+09,9E+09,9E+09]];
    CONST robtarget Target_1621:=[[403.47,280,-20],[1,0,0,0],[0,0,0,0],[9E+09,9E+09,9E+09,9E+09,9E+09,9E+09]];
    !Initializing variables
    VAR num calibrationConfermation;
    VAR errstr my_title := "Number not in system";
    VAR errstr str1 := "The number can't be drawn as it's not in the system.";
    VAR errstr str2 := "More numbers will be available in the next update.";
    VAR errstr str3 := " ";
    VAR errstr str4 := " ";
    VAR string  StringNum3;
    VAR num number1:=0;
    VAR num number2:=0;
    VAR num number3:=0;
    VAR num choice;
    var num movex:=200;
    var num movey:=100;
    VAR num len ;
    VAR num number;
    CONST robtarget Target_6290:=[[201.406869026,153.990304266,-6.388786874],[1,0.000000007,-0.000000007,-0.000000072],[-1,-1,0,0],[9E+09,9E+09,9E+09,9E+09,9E+09,9E+09]];
    CONST robtarget Target_6300:=[[201.406871282,101.150391193,-6.388740842],[1,0.000000023,-0.000000006,-0.000000107],[-1,-1,0,0],[9E+09,9E+09,9E+09,9E+09,9E+09,9E+09]];
    CONST robtarget Target_6310:=[[230.202403305,127.506100297,-6.388646383],[1,0.000000022,-0.000000006,-0.000000092],[0,-1,1,0],[9E+09,9E+09,9E+09,9E+09,9E+09,9E+09]];
    CONST robtarget Target_6320:=[[255.840299851,100.43138791,-6.388497737],[1,0.000000006,-0.000000006,-0.000000019],[0,-1,1,0],[9E+09,9E+09,9E+09,9E+09,9E+09,9E+09]];
    CONST robtarget Target_6330:=[[255.840298139,154.370706888,-6.388434501],[1,0.000000006,-0.000000006,0.000000028],[0,-1,1,0],[9E+09,9E+09,9E+09,9E+09,9E+09,9E+09]];
    !***********************************************************
    !
    ! Module:  Module1
    !
    ! Description:
    !
    !   This programme is written for the IRB 120 robot manipular with a custom built end effector that holds a standard Bic pen.
    !   The instructions provided by the programme will allow the robot to draw images with predefined targets.
    ! Author: Marlon Gwira
    !
    ! Version: 1.0
    !
    !***********************************************************


    !***********************************************************
    !
    ! Procedure main
    !
    !   This is the entry point of your program
    !
    !***********************************************************
    PROC main()
        !TPReadFK Creates function windows on the flexpendant. For information about functions for rapid please refere to the following link:
        !file:///C:/Users/Marlon%20Gwira/Downloads/RAPID%20reference%20manual.pdf
        !All the procedures are put in a while loop so it goes back to main after each task is completed
        WHILE TRUE DO
            TPReadFK choice,"Please select one of the options below","Addition","Draw all available","Draw image","Draw initials","Exit";
            IF choice=1 THEN
            addition;
                ELSEIF choice=2 THEN
                TPWrite "or would you like to calibrate the workspace before drawing images?";
                TPWrite "press 1 for YES 0 for NO";
                TPReadNum calibrationConfermation, "";
                    IF calibrationConfermation = 1 THEN
                        paperCalibration;
                        ELSEIF calibrationConfermation = 0 THEN
                            TPWrite "Drawing images";
                    ENDIF
                drawing_1;
                DRAW_INITIALS;
                ELSEIF choice=3 THEN
                drawing_1;
                ELSEIF choice=4 THEN
                DRAW_INITIALS;
                ELSEIF choice=5 THEN
                EXIT;
            ENDIF
            TPWrite "drawing complete";
            home;
            WaitTime 3;
            TPErase;
        ENDWHILE
    ENDPROC
    !The procedures below act like functions and are called back in the main
    PROC addition()
       TPErase;!this function clears the display on the Flexpendant
       TPReadNum number1, "type in number then press OK:";! Allows for numeric input in the Flexpendant
       TPReadNum number2,"type in number to add to then press OK:";
       number3 := number1+number2;
       TPWrite "the result is:"\Num:=number3;
       IF number3 = 0 THEN           !Comparing the values of the the results to the number that corresponds to the path we want to draw
           number_0;
           ELSEIF number3 = 1 THEN
               number_1;
           ELSEIF number3 = 2 THEN
               number_2;
           ELSEIF number3 = 3 THEN
               number_3;
           ELSEIF number3 = 4 THEN
               number_4;
           ELSEIF number3 = 5 THEN
               number_5;
           ELSEIF number3 = 6 THEN
               number_6;
           ELSEIF number3 = 7 THEN
               number_7;
           ELSEIF number3 = 8 THEN
               number_8;
           ELSEIF number3 = 9 THEN
               number_9;
       ENDIF
       IF number3 > 9 THEN
           ErrLog 4800, my_title, str1,str2,str3,str4;
       ENDIF
     ENDPROC

    !this procedure contains linear moves to draw a predefined image
    PROC drawing_1()
        TPErase;
        MoveL Target_1640_2,v50,z100,PenTool\WObj:=A3paper;
        MoveL Target_1641,v50,fine,PenTool\WObj:=A3paper;
        MoveL Target_1650,v50,fine,PenTool\WObj:=A3paper;
        MoveL Target_1660,v50,z100,PenTool\WObj:=A3paper;
        MoveL Target_1670,v50,z100,PenTool\WObj:=A3paper;
        MoveL Target_1680,v50,z100,PenTool\WObj:=A3paper;
        MoveL Target_1690,v50,z100,PenTool\WObj:=A3paper;
        MoveL Target_1700,v50,z100,PenTool\WObj:=A3paper;
        MoveL Target_1710,v50,z100,PenTool\WObj:=A3paper;
        MoveL Target_1720,v50,z100,PenTool\WObj:=A3paper;
        MoveL Target_1730,v50,z100,PenTool\WObj:=A3paper;
        MoveL Target_1740,v50,z100,PenTool\WObj:=A3paper;
        MoveL Target_1750,v50,z100,PenTool\WObj:=A3paper;
        MoveL Target_1760,v50,z100,PenTool\WObj:=A3paper;
        MoveL Target_1770,v50,z100,PenTool\WObj:=A3paper;
        MoveL Target_1780,v50,z100,PenTool\WObj:=A3paper;
        MoveL Target_1790,v50,z100,PenTool\WObj:=A3paper;
        MoveL Target_1800,v50,z100,PenTool\WObj:=A3paper;
        MoveL Target_1810,v50,z100,PenTool\WObj:=A3paper;
        MoveL Target_1820,v50,z100,PenTool\WObj:=A3paper;
        MoveL Target_1830,v50,z100,PenTool\WObj:=A3paper;
        MoveL Target_1840,v50,z100,PenTool\WObj:=A3paper;
        MoveL Target_1850,v50,z100,PenTool\WObj:=A3paper;
        MoveL Target_1860,v50,z100,PenTool\WObj:=A3paper;
        MoveL Target_1870,v50,z100,PenTool\WObj:=A3paper;
        MoveL Target_1880,v50,z100,PenTool\WObj:=A3paper;
        MoveL Target_1890,v50,z100,PenTool\WObj:=A3paper;
        MoveL Target_1900,v50,z100,PenTool\WObj:=A3paper;
        MoveL Target_1910,v50,z100,PenTool\WObj:=A3paper;
        MoveL Target_1920,v50,z100,PenTool\WObj:=A3paper;
        MoveL Target_1930,v50,z100,PenTool\WObj:=A3paper;
        MoveL Target_1940,v50,z100,PenTool\WObj:=A3paper;
        MoveL Target_1950,v50,z100,PenTool\WObj:=A3paper;
        MoveL Target_1960,v50,z100,PenTool\WObj:=A3paper;
        MoveL Target_1970,v50,z100,PenTool\WObj:=A3paper;
        MoveL Target_1980,v50,z100,PenTool\WObj:=A3paper;
        MoveL Target_1990,v50,z100,PenTool\WObj:=A3paper;
        MoveL Target_2000,v50,z100,PenTool\WObj:=A3paper;
        MoveL Target_2010,v50,z100,PenTool\WObj:=A3paper;
        MoveL Target_2020,v50,z100,PenTool\WObj:=A3paper;
        MoveL Target_2030,v50,z100,PenTool\WObj:=A3paper;
        MoveL Target_2040,v50,z100,PenTool\WObj:=A3paper;
        MoveL Target_2050,v50,z100,PenTool\WObj:=A3paper;
        MoveL Target_2060,v50,z100,PenTool\WObj:=A3paper;
        MoveL Target_2070,v50,z100,PenTool\WObj:=A3paper;
        MoveL Target_2080,v50,z100,PenTool\WObj:=A3paper;
        MoveL Target_2090,v50,z100,PenTool\WObj:=A3paper;
        MoveL Target_2100,v50,z100,PenTool\WObj:=A3paper;
        MoveL Target_2110,v50,z100,PenTool\WObj:=A3paper;
        MoveL Target_2120,v50,z100,PenTool\WObj:=A3paper;
        MoveL Target_2130,v50,z100,PenTool\WObj:=A3paper;
        MoveL Target_2140,v50,z100,PenTool\WObj:=A3paper;
        MoveL Target_2150,v50,z100,PenTool\WObj:=A3paper;
        MoveL Target_2160,v50,z100,PenTool\WObj:=A3paper;
        MoveL Target_2170,v50,z100,PenTool\WObj:=A3paper;
        MoveL Target_2180,v50,z100,PenTool\WObj:=A3paper;
        MoveL Target_2190,v50,z100,PenTool\WObj:=A3paper;
        MoveL Target_2200,v50,z100,PenTool\WObj:=A3paper;
        MoveL Target_2210,v50,z100,PenTool\WObj:=A3paper;
        MoveL Target_2220,v50,z100,PenTool\WObj:=A3paper;
        MoveL Target_2230,v50,z100,PenTool\WObj:=A3paper;
        MoveL Target_2240,v50,z100,PenTool\WObj:=A3paper;
        MoveL Target_2250,v50,z100,PenTool\WObj:=A3paper;
        MoveL Target_2260,v50,z100,PenTool\WObj:=A3paper;
        MoveL Target_2270,v50,z100,PenTool\WObj:=A3paper;
        MoveL Target_2280,v50,z100,PenTool\WObj:=A3paper;
        MoveL Target_2290,v50,z100,PenTool\WObj:=A3paper;
        MoveL Target_2300,v50,z100,PenTool\WObj:=A3paper;
        MoveL Target_2310,v50,z100,PenTool\WObj:=A3paper;
        MoveL Target_2320,v50,z100,PenTool\WObj:=A3paper;
        MoveL Target_2330,v50,z100,PenTool\WObj:=A3paper;
        MoveL Target_2340,v50,z100,PenTool\WObj:=A3paper;
        MoveL Target_2350,v50,z100,PenTool\WObj:=A3paper;
        MoveL Target_2360,v50,z100,PenTool\WObj:=A3paper;
        MoveL Target_2370,v50,z100,PenTool\WObj:=A3paper;
        MoveL Target_2380,v50,z100,PenTool\WObj:=A3paper;
        MoveL Target_2390,v50,z100,PenTool\WObj:=A3paper;
        MoveL Target_2400,v50,z100,PenTool\WObj:=A3paper;
        MoveL Target_2410,v50,z100,PenTool\WObj:=A3paper;
        MoveL Target_2420,v50,z100,PenTool\WObj:=A3paper;
        MoveL Target_2430,v50,z100,PenTool\WObj:=A3paper;
        MoveL Target_2440,v50,z100,PenTool\WObj:=A3paper;
        MoveL Target_2450,v50,z100,PenTool\WObj:=A3paper;
        MoveL Target_2460,v50,z100,PenTool\WObj:=A3paper;
        MoveL Target_2470,v50,z100,PenTool\WObj:=A3paper;
        MoveL Target_2480,v50,z100,PenTool\WObj:=A3paper;
        MoveL Target_2490,v50,z100,PenTool\WObj:=A3paper;
        MoveL Target_2500,v50,z100,PenTool\WObj:=A3paper;
        MoveL Target_2510,v50,z100,PenTool\WObj:=A3paper;
        MoveL Target_2520,v50,z100,PenTool\WObj:=A3paper;
        MoveL Target_2530,v50,z100,PenTool\WObj:=A3paper;
        MoveL Target_2540,v50,z100,PenTool\WObj:=A3paper;
        MoveL Target_2550,v50,z100,PenTool\WObj:=A3paper;
        MoveL Target_2560,v50,z100,PenTool\WObj:=A3paper;
        MoveL Target_2570,v50,z100,PenTool\WObj:=A3paper;
        MoveL Target_2580,v50,z100,PenTool\WObj:=A3paper;
        MoveL Target_2590,v50,z100,PenTool\WObj:=A3paper;
        MoveL Target_2600,v50,z100,PenTool\WObj:=A3paper;
        MoveL Target_2610,v50,z100,PenTool\WObj:=A3paper;
        MoveL Target_2620,v50,z100,PenTool\WObj:=A3paper;
        MoveL Target_2630,v50,z100,PenTool\WObj:=A3paper;
        MoveL Target_2640,v50,z100,PenTool\WObj:=A3paper;
        MoveL Target_2650,v50,z100,PenTool\WObj:=A3paper;
        MoveL Target_2660,v50,z100,PenTool\WObj:=A3paper;
        MoveL Target_2670,v50,z100,PenTool\WObj:=A3paper;
        MoveL Target_2680,v50,z100,PenTool\WObj:=A3paper;
        MoveL Target_2690,v50,z100,PenTool\WObj:=A3paper;
        MoveL Target_2700,v50,z100,PenTool\WObj:=A3paper;
        MoveL Target_2710,v50,z100,PenTool\WObj:=A3paper;
        MoveL Target_2720,v50,z100,PenTool\WObj:=A3paper;
        MoveL Target_2730,v50,z100,PenTool\WObj:=A3paper;
        MoveL Target_2740,v50,z100,PenTool\WObj:=A3paper;
        MoveL Target_2750,v50,z100,PenTool\WObj:=A3paper;
        MoveL Target_2760,v50,z100,PenTool\WObj:=A3paper;
        MoveL Target_2770,v50,z100,PenTool\WObj:=A3paper;
        MoveL Target_2780,v50,z100,PenTool\WObj:=A3paper;
        MoveL Target_2790,v50,z100,PenTool\WObj:=A3paper;
        MoveL Target_2800,v50,z100,PenTool\WObj:=A3paper;
        MoveL Target_2810,v50,z100,PenTool\WObj:=A3paper;
        MoveL Target_2820,v50,z100,PenTool\WObj:=A3paper;
        MoveL Target_2830,v50,z100,PenTool\WObj:=A3paper;
        MoveL Target_2840,v50,z100,PenTool\WObj:=A3paper;
        MoveL Target_2850,v50,z100,PenTool\WObj:=A3paper;
        MoveL Target_2860,v50,z100,PenTool\WObj:=A3paper;
        MoveL Target_2870,v50,z100,PenTool\WObj:=A3paper;
        MoveL Target_2880,v50,z100,PenTool\WObj:=A3paper;
        MoveL Target_2890,v50,z100,PenTool\WObj:=A3paper;
        MoveL Target_2900,v50,z100,PenTool\WObj:=A3paper;
        MoveL Target_2910,v50,z100,PenTool\WObj:=A3paper;
        MoveL Target_2920,v50,z100,PenTool\WObj:=A3paper;
        MoveL Target_2930,v50,z100,PenTool\WObj:=A3paper;
        MoveL Target_2940,v50,z100,PenTool\WObj:=A3paper;
        MoveL Target_2950,v50,z100,PenTool\WObj:=A3paper;
        MoveL Target_2960,v50,z100,PenTool\WObj:=A3paper;
        MoveL Target_2970,v50,z100,PenTool\WObj:=A3paper;
        MoveL Target_2980,v50,z100,PenTool\WObj:=A3paper;
        MoveL Target_2990,v50,z100,PenTool\WObj:=A3paper;
        MoveL Target_3000,v50,z100,PenTool\WObj:=A3paper;
        MoveL Target_3010,v50,z100,PenTool\WObj:=A3paper;
        MoveL Target_3020,v50,z100,PenTool\WObj:=A3paper;
        MoveL Target_3030,v50,z100,PenTool\WObj:=A3paper;
        MoveL Target_3040,v50,z100,PenTool\WObj:=A3paper;
        MoveL Target_3050,v50,z100,PenTool\WObj:=A3paper;
        MoveL Target_3060,v50,z100,PenTool\WObj:=A3paper;
        MoveL Target_3070,v50,z100,PenTool\WObj:=A3paper;
        MoveL Target_3080,v50,z100,PenTool\WObj:=A3paper;
        MoveL Target_3090,v50,z100,PenTool\WObj:=A3paper;
        MoveL Target_3100,v50,z100,PenTool\WObj:=A3paper;
        MoveL Target_3110,v50,z100,PenTool\WObj:=A3paper;
        MoveL Target_3120,v50,z100,PenTool\WObj:=A3paper;
        MoveL Target_3130,v50,z100,PenTool\WObj:=A3paper;
        MoveL Target_3140,v50,z100,PenTool\WObj:=A3paper;
        MoveL Target_3150,v50,z100,PenTool\WObj:=A3paper;
        MoveL Target_3160,v50,z100,PenTool\WObj:=A3paper;
        MoveL Target_3170,v50,z100,PenTool\WObj:=A3paper;
        MoveL Target_3180,v50,z100,PenTool\WObj:=A3paper;
        MoveL Target_3190,v50,z100,PenTool\WObj:=A3paper;
        MoveL Target_3200,v50,z100,PenTool\WObj:=A3paper;
        MoveL Target_3210,v50,z100,PenTool\WObj:=A3paper;
        MoveL Target_3220,v50,z100,PenTool\WObj:=A3paper;
        MoveL Target_3230,v50,z100,PenTool\WObj:=A3paper;
        MoveL Target_3240,v50,z100,PenTool\WObj:=A3paper;
        MoveL Target_3250,v50,z100,PenTool\WObj:=A3paper;
        MoveL Target_3260,v50,z100,PenTool\WObj:=A3paper;
        MoveL Target_3270,v50,z100,PenTool\WObj:=A3paper;
        MoveL Target_3280,v50,z100,PenTool\WObj:=A3paper;
        MoveL Target_3290,v50,z100,PenTool\WObj:=A3paper;
        MoveL Target_3300,v50,z100,PenTool\WObj:=A3paper;
        MoveL Target_3310,v50,z100,PenTool\WObj:=A3paper;
        MoveL Target_3320,v50,z100,PenTool\WObj:=A3paper;
        MoveL Target_3330,v50,z100,PenTool\WObj:=A3paper;
        MoveL Target_3340,v50,z100,PenTool\WObj:=A3paper;
        MoveL Target_3350,v50,z100,PenTool\WObj:=A3paper;
        MoveL Target_3360,v50,z100,PenTool\WObj:=A3paper;
        MoveL Target_3370,v50,z100,PenTool\WObj:=A3paper;
        MoveL Target_3380,v50,z100,PenTool\WObj:=A3paper;
        MoveL Target_3390,v50,z100,PenTool\WObj:=A3paper;
        MoveL Target_3400,v50,z100,PenTool\WObj:=A3paper;
        MoveL Target_3410,v50,z100,PenTool\WObj:=A3paper;
        MoveL Target_3420,v50,z100,PenTool\WObj:=A3paper;
        MoveL Target_3430,v50,z100,PenTool\WObj:=A3paper;
        MoveL Target_3440,v50,z100,PenTool\WObj:=A3paper;
        MoveL Target_3450,v50,z100,PenTool\WObj:=A3paper;
        MoveL Target_3460,v50,z100,PenTool\WObj:=A3paper;
        MoveL Target_3470,v50,z100,PenTool\WObj:=A3paper;
        MoveL Target_3480,v50,z100,PenTool\WObj:=A3paper;
        MoveL Target_3490,v50,z100,PenTool\WObj:=A3paper;
        MoveL Target_3500,v50,z100,PenTool\WObj:=A3paper;
        MoveL Target_3510,v50,z100,PenTool\WObj:=A3paper;
        MoveL Target_3520,v50,z100,PenTool\WObj:=A3paper;
        MoveL Target_3530,v50,z100,PenTool\WObj:=A3paper;
        MoveL Target_3540,v50,z100,PenTool\WObj:=A3paper;
        MoveL Target_3550,v50,z100,PenTool\WObj:=A3paper;
        MoveL Target_3560,v50,z100,PenTool\WObj:=A3paper;
        MoveL Target_3570,v50,z100,PenTool\WObj:=A3paper;
        MoveL Target_3580,v50,z100,PenTool\WObj:=A3paper;
        MoveL Target_3590,v50,z100,PenTool\WObj:=A3paper;
        MoveL Target_3600,v50,z100,PenTool\WObj:=A3paper;
        MoveL Target_3610,v50,z100,PenTool\WObj:=A3paper;
        MoveL Target_3620,v50,z100,PenTool\WObj:=A3paper;
        MoveL Target_3630,v50,z100,PenTool\WObj:=A3paper;
        MoveL Target_3640,v50,z100,PenTool\WObj:=A3paper;
        MoveL Target_3650,v50,z100,PenTool\WObj:=A3paper;
        MoveL Target_3660,v50,z100,PenTool\WObj:=A3paper;
        MoveL Target_3670,v50,z100,PenTool\WObj:=A3paper;
        MoveL Target_3680,v50,z100,PenTool\WObj:=A3paper;
        MoveL Target_3690,v50,z100,PenTool\WObj:=A3paper;
        MoveL Target_3700,v50,z100,PenTool\WObj:=A3paper;
        MoveL Target_3710,v50,z100,PenTool\WObj:=A3paper;
        MoveL Target_3720,v50,z100,PenTool\WObj:=A3paper;
        MoveL Target_3730,v50,z100,PenTool\WObj:=A3paper;
        MoveL Target_3740,v50,z100,PenTool\WObj:=A3paper;
        MoveL Target_3750,v50,fine,PenTool\WObj:=A3paper;
        MoveL Target_1640_2,v50,z100,PenTool\WObj:=A3paper;

